Yaskawa INFORM job: A_NAIHAN_0617_1_PAINT_1.JBI

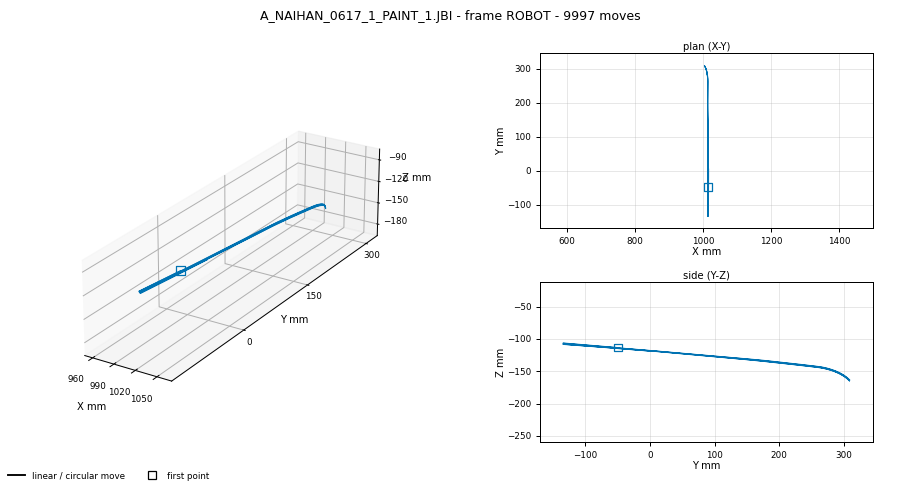
[picture p0: tool path of A_NAIHAN_0617_1_PAINT_1.JBI in frame ROBOT, 9997 of 9997 moves have a stored position in this frame; points joined in program order, loops and branches not executed]
/JOB
//NAME A_NAIHAN_0617_1_PAINT1
//POS
///NPOS 9997,0,0,0,0,0
///TOOL 1
///USER 0
///POSTYPE ROBOT
///RECTAN
///RCONF 0,0,0,0,1,0,0,0,0,0,0,0,0,0,0,0,0,0,0,0,0,0,0,0
C00000=1013.173,-49.105,-113.230,-28.110,44.378,-33.833
C00001=1013.171,-49.416,-113.204,-28.117,44.440,-33.820
C00002=1013.169,-49.806,-113.172,-28.126,44.517,-33.803
C00003=1013.167,-50.039,-113.152,-28.131,44.563,-33.794
C00004=1013.166,-50.273,-113.134,-28.136,44.610,-33.784
C00005=1013.165,-50.506,-113.114,-28.141,44.658,-33.775
C00006=1013.163,-50.741,-113.095,-28.147,44.706,-33.765
C00007=1013.162,-50.974,-113.075,-28.152,44.754,-33.754
C00008=1013.160,-51.207,-113.056,-28.157,44.802,-33.745
C00009=1013.160,-51.442,-113.037,-28.163,44.851,-33.735
C00010=1013.158,-51.675,-113.017,-28.168,44.899,-33.725
C00011=1013.156,-51.909,-112.998,-28.173,44.948,-33.715
C00012=1013.155,-52.143,-112.978,-28.179,44.998,-33.705
C00013=1013.154,-52.376,-112.959,-28.184,45.047,-33.695
C00014=1013.153,-52.610,-112.940,-28.189,45.097,-33.683
C00015=1013.151,-52.843,-112.921,-28.195,45.148,-33.674
C00016=1013.150,-53.077,-112.901,-28.200,45.199,-33.663
C00017=1013.148,-53.311,-112.882,-28.206,45.249,-33.653
C00018=1013.147,-53.544,-112.863,-28.212,45.300,-33.643
C00019=1013.146,-53.778,-112.844,-28.217,45.351,-33.632
C00020=1013.144,-54.011,-112.825,-28.223,45.403,-33.622
C00021=1013.143,-54.245,-112.804,-28.228,45.455,-33.612
C00022=1013.141,-54.479,-112.786,-28.234,45.507,-33.600
C00023=1013.140,-54.712,-112.766,-28.240,45.559,-33.590
C00024=1013.138,-54.946,-112.747,-28.245,45.612,-33.579
C00025=1013.137,-55.179,-112.728,-28.251,45.666,-33.568
C00026=1013.136,-55.414,-112.708,-28.257,45.718,-33.557
C00027=1013.134,-55.647,-112.689,-28.262,45.772,-33.547
C00028=1013.133,-55.881,-112.670,-28.268,45.825,-33.536
C00029=1013.131,-56.114,-112.651,-28.274,45.881,-33.525
C00030=1013.129,-56.348,-112.631,-28.280,45.934,-33.514
C00031=1013.129,-56.582,-112.612,-28.286,45.989,-33.503
C00032=1013.126,-56.816,-112.592,-28.292,46.045,-33.492
C00033=1013.125,-57.050,-112.573,-28.298,46.100,-33.480
C00034=1013.124,-57.284,-112.554,-28.304,46.156,-33.470
C00035=1013.122,-57.518,-112.534,-28.309,46.211,-33.459
C00036=1013.120,-57.753,-112.515,-28.315,46.268,-33.447
C00037=1013.119,-57.988,-112.495,-28.321,46.324,-33.437
C00038=1013.117,-58.222,-112.476,-28.328,46.382,-33.426
C00039=1013.116,-58.457,-112.457,-28.334,46.439,-33.414
C00040=1013.114,-58.693,-112.437,-28.340,46.496,-33.403
C00041=1013.113,-58.928,-112.418,-28.346,46.555,-33.390
C00042=1013.111,-59.163,-112.399,-28.352,46.614,-33.380
C00043=1013.110,-59.400,-112.379,-28.358,46.672,-33.368
C00044=1013.108,-59.635,-112.359,-28.364,46.732,-33.356
C00045=1013.107,-59.871,-112.340,-28.371,46.791,-33.345
C00046=1013.105,-60.108,-112.321,-28.377,46.850,-33.333
C00047=1013.103,-60.344,-112.301,-28.383,46.911,-33.322
C00048=1013.102,-60.581,-112.282,-28.390,46.972,-33.310
C00049=1013.101,-60.818,-112.262,-28.396,47.033,-33.298
C00050=1013.099,-61.055,-112.242,-28.402,47.093,-33.287
C00051=1013.097,-61.292,-112.222,-28.409,47.154,-33.275
C00052=1013.096,-61.529,-112.203,-28.415,47.217,-33.262
C00053=1013.094,-61.766,-112.183,-28.422,47.279,-33.251
C00054=1013.092,-62.005,-112.163,-28.428,47.341,-33.238
C00055=1013.090,-62.242,-112.144,-28.435,47.404,-33.227
C00056=1013.089,-62.480,-112.124,-28.441,47.467,-33.215
C00057=1013.087,-62.719,-112.104,-28.448,47.530,-33.203
C00058=1013.085,-62.957,-112.085,-28.455,47.595,-33.190
C00059=1013.083,-63.196,-112.065,-28.461,47.659,-33.178
C00060=1013.082,-63.434,-112.045,-28.468,47.723,-33.167
C00061=1013.080,-63.673,-112.025,-28.475,47.789,-33.155
C00062=1013.078,-63.913,-112.006,-28.481,47.854,-33.142
C00063=1013.077,-64.151,-111.986,-28.488,47.919,-33.130
C00064=1013.075,-64.391,-111.966,-28.495,47.985,-33.118
C00065=1013.073,-64.630,-111.946,-28.502,48.051,-33.105
C00066=1013.072,-64.870,-111.927,-28.508,48.117,-33.093
C00067=1013.070,-65.109,-111.907,-28.515,48.185,-33.081
C00068=1013.068,-65.349,-111.887,-28.522,48.252,-33.068
C00069=1013.067,-65.589,-111.867,-28.529,48.319,-33.056
C00070=1013.065,-65.829,-111.848,-28.536,48.387,-33.043
C00071=1013.062,-66.069,-111.827,-28.543,48.456,-33.030
C00072=1013.061,-66.309,-111.807,-28.550,48.524,-33.019
C00073=1013.059,-66.549,-111.787,-28.557,48.593,-33.005
C00074=1013.057,-66.790,-111.767,-28.564,48.662,-32.993
C00075=1013.056,-67.030,-111.747,-28.571,48.732,-32.980
C00076=1013.054,-67.270,-111.728,-28.578,48.802,-32.968
C00077=1013.052,-67.511,-111.707,-28.585,48.871,-32.956
C00078=1013.050,-67.752,-111.688,-28.593,48.941,-32.944
C00079=1013.049,-67.992,-111.668,-28.600,49.012,-32.931
C00080=1013.046,-68.233,-111.648,-28.607,49.083,-32.918
C00081=1013.044,-68.473,-111.628,-28.614,49.155,-32.905
C00082=1013.043,-68.713,-111.608,-28.621,49.227,-32.893
C00083=1013.040,-68.954,-111.588,-28.629,49.298,-32.880
C00084=1013.039,-69.195,-111.568,-28.636,49.371,-32.869
C00085=1013.037,-69.435,-111.549,-28.643,49.443,-32.855
C00086=1013.036,-69.676,-111.528,-28.650,49.516,-32.842
C00087=1013.033,-69.917,-111.509,-28.658,49.589,-32.830
C00088=1013.031,-70.158,-111.488,-28.665,49.662,-32.818
C00089=1013.030,-70.398,-111.469,-28.673,49.736,-32.805
C00090=1013.028,-70.639,-111.448,-28.680,49.811,-32.792
C00091=1013.026,-70.880,-111.429,-28.688,49.884,-32.779
C00092=1013.024,-71.110,-111.409,-28.695,49.956,-32.767
C00093=1013.022,-71.340,-111.390,-28.702,50.028,-32.756
C00094=1013.020,-71.601,-111.369,-28.710,50.110,-32.742
C00095=1013.019,-71.842,-111.349,-28.718,50.185,-32.729
C00096=1013.016,-72.082,-111.329,-28.725,50.261,-32.717
C00097=1013.014,-72.323,-111.309,-28.733,50.338,-32.703
C00098=1013.013,-72.563,-111.289,-28.741,50.414,-32.691
C00099=1013.010,-72.804,-111.269,-28.748,50.491,-32.678
C00100=1013.009,-73.044,-111.250,-28.756,50.567,-32.667
C00101=1013.007,-73.284,-111.229,-28.764,50.644,-32.653
C00102=1013.005,-73.524,-111.209,-28.771,50.722,-32.641
C00103=1013.003,-73.764,-111.189,-28.779,50.799,-32.628
C00104=1013.000,-74.004,-111.169,-28.787,50.879,-32.615
C00105=1012.999,-74.244,-111.149,-28.795,50.956,-32.603
C00106=1012.997,-74.484,-111.130,-28.803,51.036,-32.590
C00107=1012.995,-74.724,-111.109,-28.810,51.114,-32.578
C00108=1012.993,-74.964,-111.090,-28.818,51.193,-32.565
C00109=1012.991,-75.204,-111.070,-28.826,51.273,-32.553
C00110=1012.989,-75.443,-111.050,-28.834,51.353,-32.541
C00111=1012.987,-75.684,-111.030,-28.842,51.434,-32.527
C00112=1012.985,-75.924,-111.009,-28.850,51.514,-32.515
C00113=1012.983,-76.163,-110.990,-28.858,51.595,-32.502
C00114=1012.981,-76.403,-110.970,-28.866,51.675,-32.490
C00115=1012.979,-76.643,-110.950,-28.874,51.756,-32.478
C00116=1012.977,-76.882,-110.930,-28.882,51.838,-32.466
C00117=1012.975,-77.122,-110.910,-28.890,51.920,-32.454
C00118=1012.973,-77.360,-110.891,-28.899,52.002,-32.442
C00119=1012.971,-77.599,-110.871,-28.907,52.084,-32.428
C00120=1012.969,-77.839,-110.850,-28.915,52.167,-32.417
C00121=1012.967,-78.077,-110.831,-28.923,52.249,-32.403
C00122=1012.965,-78.316,-110.810,-28.931,52.333,-32.391
C00123=1012.963,-78.555,-110.791,-28.940,52.416,-32.381
C00124=1012.961,-78.794,-110.771,-28.948,52.499,-32.368
C00125=1012.959,-79.032,-110.751,-28.956,52.584,-32.355
C00126=1012.957,-79.271,-110.732,-28.965,52.668,-32.343
C00127=1012.955,-79.509,-110.711,-28.973,52.752,-32.332
C00128=1012.953,-79.747,-110.692,-28.981,52.837,-32.319
C00129=1012.951,-79.985,-110.672,-28.990,52.921,-32.308
C00130=1012.949,-80.222,-110.652,-28.998,53.006,-32.295
C00131=1012.947,-80.460,-110.632,-29.007,53.092,-32.283
C00132=1012.945,-80.697,-110.613,-29.015,53.177,-32.271
C00133=1012.943,-80.934,-110.593,-29.024,53.263,-32.259
C00134=1012.941,-81.169,-110.573,-29.032,53.348,-32.248
C00135=1012.939,-81.406,-110.554,-29.041,53.434,-32.236
C00136=1012.937,-81.643,-110.534,-29.049,53.520,-32.225
C00137=1012.935,-81.880,-110.514,-29.058,53.607,-32.213
C00138=1012.933,-82.117,-110.495,-29.067,53.695,-32.201
C00139=1012.930,-82.354,-110.475,-29.075,53.782,-32.190
C00140=1012.928,-82.591,-110.455,-29.084,53.870,-32.178
C00141=1012.927,-82.827,-110.435,-29.093,53.957,-32.166
C00142=1012.924,-83.062,-110.416,-29.102,54.045,-32.156
C00143=1012.922,-83.298,-110.395,-29.110,54.133,-32.144
C00144=1012.921,-83.535,-110.376,-29.119,54.222,-32.132
C00145=1012.918,-83.770,-110.357,-29.128,54.310,-32.122
C00146=1012.916,-84.002,-110.337,-29.137,54.397,-32.110
C00147=1012.914,-84.234,-110.318,-29.146,54.485,-32.100
C00148=1012.912,-84.468,-110.298,-29.155,54.574,-32.089
C00149=1012.910,-84.708,-110.278,-29.164,54.666,-32.077
C00150=1012.908,-84.964,-110.257,-29.174,54.764,-32.066
C00151=1012.905,-85.239,-110.234,-29.184,54.869,-32.052
C00152=1012.903,-85.524,-110.210,-29.195,54.978,-32.039
C00153=1012.900,-85.807,-110.187,-29.206,55.087,-32.027
C00154=1012.898,-86.076,-110.164,-29.217,55.192,-32.014
C00155=1012.895,-86.327,-110.142,-29.227,55.290,-32.003
C00156=1012.894,-86.561,-110.123,-29.236,55.382,-31.992
C00157=1012.892,-86.793,-110.104,-29.245,55.471,-31.982
C00158=1012.889,-87.101,-110.078,-29.258,55.593,-31.968
C00159=1012.886,-87.464,-110.048,-29.272,55.737,-31.952
C00160=1012.884,-87.683,-110.030,-29.281,55.823,-31.942
C00161=1012.882,-87.899,-110.012,-29.290,55.908,-31.933
C00162=1012.880,-88.115,-109.993,-29.299,55.995,-31.924
C00163=1012.878,-88.341,-109.975,-29.308,56.085,-31.914
C00164=1012.875,-88.568,-109.956,-29.317,56.176,-31.905
C00165=1012.874,-88.801,-109.936,-29.327,56.270,-31.895
C00166=1012.871,-89.068,-109.913,-29.338,56.377,-31.883
C00167=1012.869,-89.365,-109.889,-29.351,56.498,-31.872
C00168=1012.866,-89.673,-109.863,-29.364,56.623,-31.858
C00169=1012.863,-89.974,-109.838,-29.376,56.745,-31.846
C00170=1012.861,-90.252,-109.814,-29.388,56.859,-31.835
C00171=1012.857,-90.648,-109.782,-29.406,57.022,-31.820
C00172=1012.855,-90.945,-109.757,-29.418,57.144,-31.807
C00173=1012.853,-91.195,-109.736,-29.429,57.248,-31.797
C00174=1012.851,-91.427,-109.716,-29.439,57.344,-31.789
C00175=1012.849,-91.658,-109.697,-29.449,57.441,-31.780
C00176=1012.847,-91.889,-109.677,-29.460,57.536,-31.771
C00177=1012.844,-92.120,-109.658,-29.470,57.633,-31.762
C00178=1012.842,-92.352,-109.639,-29.480,57.730,-31.753
C00179=1012.840,-92.582,-109.620,-29.491,57.828,-31.745
C00180=1012.838,-92.812,-109.600,-29.501,57.925,-31.737
C00181=1012.837,-93.042,-109.581,-29.511,58.022,-31.728
C00182=1012.834,-93.271,-109.561,-29.522,58.119,-31.721
C00183=1012.831,-93.501,-109.542,-29.533,58.217,-31.713
C00184=1012.830,-93.730,-109.523,-29.543,58.315,-31.703
C00185=1012.828,-93.959,-109.504,-29.554,58.412,-31.696
C00186=1012.826,-94.188,-109.485,-29.565,58.510,-31.689
C00187=1012.824,-94.416,-109.465,-29.575,58.608,-31.681
C00188=1012.821,-94.643,-109.447,-29.586,58.706,-31.674
C00189=1012.819,-94.871,-109.427,-29.597,58.805,-31.666
C00190=1012.817,-95.097,-109.408,-29.608,58.902,-31.659
C00191=1012.816,-95.323,-109.389,-29.619,59.001,-31.652
C00192=1012.814,-95.549,-109.370,-29.630,59.100,-31.645
C00193=1012.812,-95.774,-109.351,-29.641,59.197,-31.638
C00194=1012.810,-95.999,-109.332,-29.652,59.297,-31.632
C00195=1012.807,-96.224,-109.313,-29.663,59.395,-31.625
C00196=1012.806,-96.448,-109.294,-29.674,59.494,-31.618
C00197=1012.804,-96.673,-109.275,-29.685,59.592,-31.611
C00198=1012.802,-96.896,-109.257,-29.697,59.692,-31.605
C00199=1012.799,-97.121,-109.238,-29.708,59.791,-31.599
C00200=1012.798,-97.345,-109.219,-29.720,59.890,-31.594
C00201=1012.796,-97.568,-109.200,-29.732,59.990,-31.589
C00202=1012.794,-97.791,-109.182,-29.743,60.090,-31.582
C00203=1012.792,-98.015,-109.162,-29.755,60.189,-31.577
C00204=1012.790,-98.239,-109.144,-29.766,60.289,-31.571
C00205=1012.788,-98.462,-109.125,-29.778,60.390,-31.566
C00206=1012.786,-98.686,-109.106,-29.790,60.491,-31.560
C00207=1012.784,-98.910,-109.088,-29.802,60.591,-31.555
C00208=1012.782,-99.134,-109.068,-29.814,60.693,-31.551
C00209=1012.780,-99.358,-109.050,-29.827,60.795,-31.545
C00210=1012.778,-99.582,-109.030,-29.839,60.896,-31.542
C00211=1012.776,-99.807,-109.011,-29.851,60.999,-31.537
C00212=1012.774,-100.080,-108.988,-29.866,61.123,-31.531
C00213=1012.770,-100.484,-108.955,-29.889,61.308,-31.523
C00214=1012.768,-100.710,-108.936,-29.902,61.411,-31.520
C00215=1012.766,-100.937,-108.916,-29.915,61.515,-31.515
C00216=1012.764,-101.163,-108.898,-29.928,61.620,-31.512
C00217=1012.762,-101.391,-108.878,-29.942,61.725,-31.509
C00218=1012.760,-101.619,-108.859,-29.955,61.831,-31.505
C00219=1012.758,-101.846,-108.839,-29.968,61.937,-31.501
C00220=1012.756,-102.075,-108.820,-29.982,62.042,-31.499
C00221=1012.754,-102.303,-108.801,-29.995,62.148,-31.496
C00222=1012.752,-102.533,-108.782,-30.009,62.256,-31.492
C00223=1012.750,-102.762,-108.762,-30.023,62.363,-31.491
C00224=1012.748,-102.992,-108.743,-30.037,62.471,-31.488
C00225=1012.746,-103.221,-108.724,-30.052,62.577,-31.486
C00226=1012.745,-103.451,-108.704,-30.066,62.686,-31.484
C00227=1012.742,-103.681,-108.685,-30.080,62.794,-31.482
C00228=1012.740,-103.912,-108.666,-30.095,62.903,-31.479
C00229=1012.738,-104.142,-108.646,-30.110,63.012,-31.479
C00230=1012.737,-104.372,-108.627,-30.125,63.121,-31.477
C00231=1012.734,-104.603,-108.607,-30.140,63.231,-31.476
C00232=1012.732,-104.835,-108.588,-30.155,63.341,-31.475
C00233=1012.730,-105.066,-108.568,-30.170,63.451,-31.474
C00234=1012.729,-105.296,-108.549,-30.186,63.561,-31.474
C00235=1012.727,-105.528,-108.529,-30.201,63.671,-31.474
C00236=1012.724,-105.760,-108.509,-30.217,63.783,-31.473
C00237=1012.722,-105.991,-108.489,-30.233,63.893,-31.475
C00238=1012.721,-106.223,-108.470,-30.249,64.005,-31.475
C00239=1012.718,-106.458,-108.450,-30.266,64.119,-31.476
C00240=1012.716,-106.700,-108.430,-30.283,64.236,-31.476
C00241=1012.714,-106.952,-108.408,-30.301,64.358,-31.478
C00242=1012.712,-107.215,-108.386,-30.320,64.486,-31.480
C00243=1012.710,-107.485,-108.363,-30.340,64.617,-31.481
C00244=1012.708,-107.760,-108.340,-30.360,64.750,-31.484
C00245=1012.705,-108.036,-108.317,-30.381,64.885,-31.486
C00246=1012.703,-108.311,-108.294,-30.402,65.020,-31.489
C00247=1012.701,-108.579,-108.270,-30.422,65.151,-31.492
C00248=1012.698,-108.839,-108.249,-30.442,65.279,-31.494
C00249=1012.697,-109.090,-108.227,-30.462,65.403,-31.498
C00250=1012.694,-109.330,-108.207,-30.482,65.521,-31.504
C00251=1012.693,-109.564,-108.188,-30.501,65.636,-31.508
C00252=1012.692,-109.795,-108.168,-30.519,65.751,-31.512
C00253=1012.689,-110.026,-108.148,-30.538,65.866,-31.517
C00254=1012.687,-110.258,-108.129,-30.558,65.981,-31.522
C00255=1012.686,-110.489,-108.109,-30.577,66.096,-31.527
C00256=1012.684,-110.721,-108.089,-30.597,66.212,-31.532
C00257=1012.682,-110.952,-108.069,-30.617,66.327,-31.538
C00258=1012.680,-111.183,-108.050,-30.637,66.444,-31.544
C00259=1012.678,-111.483,-108.024,-30.664,66.593,-31.553
C00260=1012.675,-111.878,-107.991,-30.699,66.792,-31.564
C00261=1012.672,-112.109,-107.971,-30.720,66.908,-31.572
C00262=1012.671,-112.340,-107.952,-30.741,67.024,-31.579
C00263=1012.669,-112.571,-107.932,-30.763,67.142,-31.587
C00264=1012.667,-112.803,-107.913,-30.784,67.259,-31.596
C00265=1012.666,-113.035,-107.893,-30.807,67.377,-31.604
C00266=1012.663,-113.266,-107.873,-30.829,67.494,-31.615
C00267=1012.662,-113.497,-107.854,-30.852,67.612,-31.624
C00268=1012.660,-113.728,-107.834,-30.875,67.730,-31.634
C00269=1012.658,-113.959,-107.815,-30.898,67.848,-31.644
C00270=1012.657,-114.190,-107.795,-30.922,67.965,-31.654
C00271=1012.655,-114.422,-107.775,-30.945,68.085,-31.665
C00272=1012.653,-114.653,-107.756,-30.970,68.203,-31.677
C00273=1012.651,-114.885,-107.736,-30.994,68.322,-31.687
C00274=1012.650,-115.115,-107.716,-31.018,68.441,-31.699
C00275=1012.648,-115.347,-107.697,-31.044,68.561,-31.713
C00276=1012.646,-115.578,-107.677,-31.070,68.680,-31.727
C00277=1012.644,-115.809,-107.658,-31.095,68.800,-31.738
C00278=1012.642,-116.040,-107.637,-31.121,68.919,-31.753
C00279=1012.641,-116.271,-107.619,-31.148,69.039,-31.769
C00280=1012.639,-116.503,-107.598,-31.175,69.160,-31.783
C00281=1012.637,-116.734,-107.579,-31.202,69.281,-31.798
C00282=1012.636,-116.965,-107.559,-31.230,69.400,-31.814
C00283=1012.635,-117.196,-107.540,-31.258,69.521,-31.830
C00284=1012.632,-117.427,-107.520,-31.286,69.642,-31.848
C00285=1012.631,-117.659,-107.500,-31.314,69.764,-31.863
C00286=1012.629,-117.890,-107.481,-31.344,69.885,-31.881
C00287=1012.628,-118.121,-107.461,-31.374,70.006,-31.900
C00288=1012.626,-118.352,-107.441,-31.404,70.128,-31.918
C00289=1012.624,-118.584,-107.422,-31.434,70.250,-31.937
C00290=1012.623,-118.814,-107.402,-31.465,70.373,-31.958
C00291=1012.621,-119.046,-107.383,-31.496,70.495,-31.977
C00292=1012.619,-119.277,-107.363,-31.529,70.617,-31.999
C00293=1012.618,-119.507,-107.343,-31.562,70.740,-32.021
C00294=1012.616,-119.739,-107.324,-31.593,70.862,-32.041
C00295=1012.615,-119.970,-107.303,-31.628,70.985,-32.066
C00296=1012.613,-120.201,-107.284,-31.662,71.109,-32.089
C00297=1012.611,-120.432,-107.265,-31.696,71.232,-32.112
C00298=1012.610,-120.663,-107.245,-31.731,71.356,-32.138
C00299=1012.608,-120.894,-107.225,-31.766,71.479,-32.162
C00300=1012.607,-121.126,-107.206,-31.803,71.603,-32.189
C00301=1012.605,-121.356,-107.186,-31.839,71.728,-32.215
C00302=1012.604,-121.588,-107.167,-31.877,71.851,-32.243
C00303=1012.602,-121.885,-107.141,-31.925,72.012,-32.278
C00304=1012.600,-122.280,-107.107,-31.992,72.225,-32.329
C00305=1012.598,-122.511,-107.087,-32.033,72.351,-32.360
///RCONF 0,0,0,0,0,0,0,0,0,0,0,0,0,0,0,0,0,0,0,0,0,0,0,0
C00306=1012.597,-122.742,-107.068,-32.073,72.475,-32.390
C00307=1012.595,-122.973,-107.048,-32.114,72.600,-32.423
C00308=1012.594,-123.204,-107.029,-32.156,72.726,-32.454
C00309=1012.592,-123.435,-107.009,-32.199,72.851,-32.489
C00310=1012.591,-123.666,-106.990,-32.242,72.976,-32.522
C00311=1012.589,-123.897,-106.970,-32.286,73.102,-32.557
C00312=1012.588,-124.128,-106.951,-32.331,73.229,-32.594
C00313=1012.586,-124.360,-106.930,-32.377,73.354,-32.630
C00314=1012.585,-124.590,-106.911,-32.424,73.480,-32.669
C00315=1012.584,-124.822,-106.891,-32.471,73.606,-32.707
C00316=1012.582,-125.052,-106.872,-32.519,73.733,-32.746
C00317=1012.581,-125.284,-106.852,-32.568,73.859,-32.788
C00318=1012.580,-125.514,-106.832,-32.618,73.986,-32.830
C00319=1012.578,-125.745,-106.813,-32.669,74.113,-32.872
C00320=1012.577,-125.976,-106.793,-32.720,74.239,-32.915
C00321=1012.575,-126.207,-106.774,-32.773,74.366,-32.960
C00322=1012.574,-126.438,-106.754,-32.827,74.493,-33.007
C00323=1012.573,-126.669,-106.734,-32.882,74.620,-33.054
C00324=1012.571,-126.900,-106.715,-32.939,74.747,-33.103
C00325=1012.570,-127.132,-106.695,-32.995,74.874,-33.151
C00326=1012.569,-127.362,-106.675,-33.053,75.002,-33.201
C00327=1012.567,-127.592,-106.655,-33.113,75.129,-33.255
C00328=1012.566,-127.824,-106.636,-33.173,75.257,-33.308
C00329=1012.565,-128.055,-106.616,-33.235,75.385,-33.363
C00330=1012.564,-128.285,-106.597,-33.297,75.514,-33.417
C00331=1012.562,-128.517,-106.577,-33.361,75.641,-33.474
C00332=1012.562,-128.748,-106.557,-33.427,75.770,-33.535
C00333=1012.560,-128.978,-106.538,-33.493,75.898,-33.593
C00334=1012.559,-129.210,-106.518,-33.562,76.027,-33.655
C00335=1012.558,-129.440,-106.498,-33.633,76.155,-33.721
C00336=1012.556,-129.671,-106.479,-33.704,76.284,-33.786
C00337=1012.555,-129.902,-106.459,-33.775,76.413,-33.849
C00338=1012.554,-130.134,-106.439,-33.850,76.541,-33.918
C00339=1012.553,-130.364,-106.419,-33.926,76.670,-33.988
C00340=1012.552,-130.595,-106.401,-34.004,76.800,-34.061
C00341=1012.551,-130.825,-106.381,-34.084,76.929,-34.135
C00342=1012.550,-131.057,-106.361,-34.164,77.058,-34.209
C00343=1012.549,-131.288,-106.341,-34.248,77.188,-34.288
C00344=1012.547,-131.603,-106.314,-34.364,77.365,-34.396
C00345=1012.545,-131.980,-106.283,-34.508,77.577,-34.531
C00346=1012.545,-132.211,-106.263,-34.600,77.706,-34.619
C00347=1012.543,-132.443,-106.243,-34.693,77.837,-34.706
C00348=1012.542,-132.673,-106.224,-34.789,77.966,-34.798
C00349=1012.541,-132.904,-106.204,-34.887,78.096,-34.891
C00350=1012.540,-133.135,-106.184,-34.989,78.227,-34.988
C00351=1012.539,-133.366,-106.165,-35.090,78.357,-35.084
C00352=1012.538,-133.596,-106.145,-35.195,78.487,-35.184
C00353=1012.537,-133.827,-106.126,-35.304,78.618,-35.290
C00354=1012.536,-134.058,-106.106,-35.416,78.749,-35.397
///RCONF 0,0,0,0,1,0,0,0,0,0,0,0,0,0,0,0,0,0,0,0,0,0,0,0
C00355=1012.642,-134.083,-106.545,-31.212,69.079,-31.891
C00356=1012.643,-133.853,-106.565,-31.181,68.940,-31.876
C00357=1012.645,-133.622,-106.584,-31.151,68.800,-31.861
C00358=1012.648,-133.391,-106.604,-31.121,68.662,-31.846
C00359=1012.649,-133.161,-106.623,-31.091,68.523,-31.831
C00360=1012.652,-132.930,-106.643,-31.063,68.383,-31.818
C00361=1012.654,-132.698,-106.662,-31.034,68.245,-31.804
C00362=1012.655,-132.468,-106.681,-31.006,68.107,-31.792
C00363=1012.658,-132.237,-106.701,-30.978,67.968,-31.779
C00364=1012.659,-132.006,-106.722,-30.950,67.831,-31.767
C00365=1012.662,-131.775,-106.742,-30.923,67.692,-31.756
C00366=1012.663,-131.544,-106.760,-30.896,67.555,-31.745
C00367=1012.665,-131.313,-106.780,-30.870,67.417,-31.736
C00368=1012.668,-131.082,-106.800,-30.844,67.280,-31.727
C00369=1012.670,-130.851,-106.820,-30.818,67.142,-31.717
C00370=1012.672,-130.621,-106.839,-30.793,67.005,-31.707
C00371=1012.674,-130.390,-106.858,-30.768,66.868,-31.700
C00372=1012.676,-130.167,-106.878,-30.744,66.735,-31.693
C00373=1012.678,-129.928,-106.898,-30.719,66.594,-31.686
C00374=1012.680,-129.698,-106.917,-30.695,66.458,-31.678
C00375=1012.682,-129.467,-106.937,-30.671,66.321,-31.672
C00376=1012.685,-129.235,-106.956,-30.648,66.185,-31.666
C00377=1012.687,-129.005,-106.976,-30.624,66.049,-31.659
C00378=1012.690,-128.774,-106.995,-30.602,65.913,-31.654
C00379=1012.692,-128.543,-107.015,-30.579,65.778,-31.650
C00380=1012.694,-128.312,-107.035,-30.556,65.641,-31.645
C00381=1012.696,-128.081,-107.054,-30.534,65.506,-31.641
C00382=1012.698,-127.850,-107.074,-30.513,65.370,-31.638
C00383=1012.700,-127.619,-107.094,-30.491,65.236,-31.635
C00384=1012.702,-127.388,-107.113,-30.470,65.100,-31.633
C00385=1012.704,-127.157,-107.132,-30.449,64.965,-31.629
C00386=1012.707,-126.926,-107.152,-30.428,64.831,-31.627
C00387=1012.709,-126.695,-107.172,-30.407,64.697,-31.626
C00388=1012.711,-126.465,-107.191,-30.387,64.562,-31.624
C00389=1012.714,-126.234,-107.211,-30.366,64.428,-31.623
C00390=1012.716,-126.003,-107.230,-30.347,64.293,-31.622
C00391=1012.718,-125.772,-107.250,-30.327,64.160,-31.623
C00392=1012.720,-125.541,-107.270,-30.307,64.026,-31.622
C00393=1012.723,-125.310,-107.289,-30.288,63.892,-31.623
C00394=1012.725,-125.078,-107.308,-30.269,63.759,-31.623
C00395=1012.728,-124.848,-107.328,-30.250,63.626,-31.624
C00396=1012.730,-124.617,-107.348,-30.231,63.493,-31.625
C00397=1012.732,-124.386,-107.367,-30.213,63.360,-31.627
C00398=1012.735,-124.155,-107.387,-30.194,63.227,-31.629
C00399=1012.737,-123.923,-107.406,-30.176,63.094,-31.631
C00400=1012.739,-123.692,-107.426,-30.158,62.961,-31.633
C00401=1012.742,-123.462,-107.445,-30.140,62.830,-31.636
C00402=1012.744,-123.231,-107.465,-30.122,62.697,-31.640
C00403=1012.746,-122.999,-107.484,-30.104,62.565,-31.642
C00404=1012.749,-122.769,-107.504,-30.087,62.434,-31.645
C00405=1012.752,-122.538,-107.523,-30.070,62.303,-31.650
C00406=1012.754,-122.307,-107.543,-30.053,62.170,-31.655
C00407=1012.756,-122.075,-107.562,-30.035,62.040,-31.658
C00408=1012.758,-121.845,-107.582,-30.019,61.909,-31.663
C00409=1012.760,-121.614,-107.602,-30.002,61.777,-31.668
C00410=1012.764,-121.383,-107.621,-29.986,61.646,-31.674
C00411=1012.766,-121.152,-107.640,-29.969,61.516,-31.679
C00412=1012.768,-120.921,-107.660,-29.953,61.385,-31.685
C00413=1012.772,-120.573,-107.689,-29.929,61.189,-31.694
C00414=1012.776,-120.227,-107.719,-29.905,60.995,-31.703
C00415=1012.778,-119.996,-107.738,-29.889,60.866,-31.710
C00416=1012.781,-119.765,-107.758,-29.873,60.736,-31.717
C00417=1012.783,-119.534,-107.777,-29.858,60.606,-31.724
C00418=1012.785,-119.303,-107.797,-29.842,60.477,-31.732
C00419=1012.788,-119.072,-107.816,-29.827,60.348,-31.739
C00420=1012.790,-118.841,-107.835,-29.812,60.219,-31.748
C00421=1012.793,-118.610,-107.855,-29.797,60.091,-31.756
C00422=1012.796,-118.378,-107.875,-29.782,59.962,-31.765
C00423=1012.799,-118.148,-107.894,-29.767,59.834,-31.774
C00424=1012.801,-117.916,-107.913,-29.752,59.705,-31.782
C00425=1012.803,-117.685,-107.933,-29.737,59.577,-31.791
C00426=1012.806,-117.455,-107.952,-29.723,59.450,-31.801
C00427=1012.808,-117.223,-107.972,-29.708,59.323,-31.809
C00428=1012.811,-116.991,-107.992,-29.694,59.195,-31.820
C00429=1012.814,-116.761,-108.011,-29.679,59.068,-31.828
C00430=1012.816,-116.529,-108.030,-29.665,58.941,-31.839
C00431=1012.818,-116.298,-108.050,-29.651,58.814,-31.849
C00432=1012.821,-116.068,-108.069,-29.637,58.688,-31.860
C00433=1012.824,-115.836,-108.089,-29.623,58.562,-31.870
C00434=1012.826,-115.605,-108.108,-29.609,58.436,-31.882
C00435=1012.829,-115.373,-108.127,-29.596,58.310,-31.893
C00436=1012.831,-115.143,-108.147,-29.582,58.185,-31.904
C00437=1012.834,-114.911,-108.167,-29.568,58.059,-31.916
C00438=1012.837,-114.680,-108.185,-29.555,57.934,-31.927
C00439=1012.839,-114.449,-108.205,-29.541,57.810,-31.938
C00440=1012.842,-114.217,-108.226,-29.528,57.685,-31.950
C00441=1012.845,-113.986,-108.244,-29.514,57.561,-31.962
C00442=1012.847,-113.755,-108.264,-29.501,57.437,-31.974
C00443=1012.850,-113.524,-108.282,-29.488,57.313,-31.988
C00444=1012.853,-113.292,-108.303,-29.475,57.189,-32.000
C00445=1012.855,-113.061,-108.322,-29.462,57.066,-32.013
C00446=1012.858,-112.830,-108.341,-29.449,56.943,-32.026
C00447=1012.861,-112.598,-108.361,-29.436,56.820,-32.040
C00448=1012.863,-112.367,-108.380,-29.423,56.697,-32.053
C00449=1012.866,-112.136,-108.399,-29.410,56.574,-32.066
C00450=1012.868,-111.904,-108.419,-29.398,56.452,-32.080
C00451=1012.871,-111.673,-108.438,-29.384,56.330,-32.092
C00452=1012.873,-111.442,-108.457,-29.372,56.208,-32.107
C00453=1012.876,-111.210,-108.477,-29.359,56.086,-32.121
C00454=1012.879,-110.979,-108.496,-29.347,55.966,-32.136
C00455=1012.882,-110.747,-108.516,-29.334,55.845,-32.149
C00456=1012.886,-110.380,-108.547,-29.315,55.653,-32.173
C00457=1012.890,-110.053,-108.573,-29.297,55.483,-32.193
C00458=1012.893,-109.822,-108.593,-29.285,55.363,-32.208
C00459=1012.895,-109.590,-108.613,-29.273,55.243,-32.224
C00460=1012.898,-109.357,-108.633,-29.260,55.121,-32.238
C00461=1012.901,-109.117,-108.652,-29.247,54.998,-32.254
C00462=1012.904,-108.866,-108.673,-29.234,54.870,-32.270
C00463=1012.907,-108.606,-108.695,-29.221,54.736,-32.289
C00464=1012.910,-108.337,-108.717,-29.207,54.599,-32.306
C00465=1012.913,-108.064,-108.741,-29.193,54.458,-32.325
C00466=1012.917,-107.787,-108.764,-29.179,54.317,-32.346
C00467=1012.920,-107.512,-108.787,-29.164,54.177,-32.364
C00468=1012.923,-107.242,-108.809,-29.151,54.040,-32.385
C00469=1012.926,-106.979,-108.831,-29.137,53.907,-32.403
C00470=1012.929,-106.727,-108.852,-29.125,53.780,-32.421
C00471=1012.932,-106.484,-108.872,-29.112,53.657,-32.438
C00472=1012.935,-106.249,-108.892,-29.100,53.539,-32.456
C00473=1012.937,-106.018,-108.911,-29.089,53.423,-32.472
C00474=1012.940,-105.786,-108.930,-29.077,53.307,-32.490
C00475=1012.943,-105.555,-108.950,-29.065,53.191,-32.507
C00476=1012.945,-105.324,-108.969,-29.054,53.076,-32.524
C00477=1012.949,-105.093,-108.988,-29.042,52.961,-32.541
C00478=1012.951,-104.861,-109.007,-29.031,52.847,-32.559
C00479=1012.954,-104.630,-109.027,-29.019,52.732,-32.576
C00480=1012.957,-104.400,-109.046,-29.008,52.618,-32.595
C00481=1012.959,-104.169,-109.066,-28.997,52.504,-32.613
C00482=1012.961,-103.939,-109.085,-28.985,52.391,-32.630
C00483=1012.964,-103.708,-109.104,-28.974,52.278,-32.648
C00484=1012.967,-103.479,-109.123,-28.963,52.166,-32.666
C00485=1012.970,-103.248,-109.142,-28.951,52.053,-32.684
C00486=1012.973,-103.019,-109.162,-28.940,51.941,-32.702
C00487=1012.975,-102.789,-109.180,-28.929,51.829,-32.721
C00488=1012.979,-102.560,-109.199,-28.918,51.718,-32.739
C00489=1012.981,-102.331,-109.219,-28.907,51.607,-32.757
C00490=1012.984,-102.102,-109.238,-28.896,51.497,-32.776
C00491=1012.986,-101.874,-109.257,-28.884,51.386,-32.795
C00492=1012.989,-101.646,-109.275,-28.873,51.276,-32.814
C00493=1012.992,-101.418,-109.294,-28.863,51.168,-32.832
C00494=1012.995,-101.191,-109.313,-28.851,51.059,-32.850
C00495=1012.997,-100.964,-109.332,-28.841,50.949,-32.870
C00496=1013.000,-100.737,-109.351,-28.830,50.843,-32.889
C00497=1013.002,-100.511,-109.370,-28.819,50.734,-32.908
C00498=1013.005,-100.285,-109.388,-28.808,50.627,-32.926
C00499=1013.008,-100.060,-109.407,-28.797,50.520,-32.946
C00500=1013.010,-99.834,-109.426,-28.787,50.414,-32.965
C00501=1013.013,-99.610,-109.445,-28.776,50.309,-32.983
C00502=1013.016,-99.385,-109.463,-28.765,50.203,-33.003
C00503=1013.020,-99.061,-109.490,-28.750,50.051,-33.031
C00504=1013.024,-98.713,-109.518,-28.733,49.888,-33.061
C00505=1013.026,-98.489,-109.537,-28.723,49.784,-33.080
C00506=1013.029,-98.266,-109.556,-28.712,49.680,-33.100
C00507=1013.032,-98.042,-109.574,-28.702,49.577,-33.119
C00508=1013.034,-97.819,-109.593,-28.691,49.473,-33.138
C00509=1013.037,-97.595,-109.611,-28.680,49.370,-33.157
C00510=1013.040,-97.372,-109.630,-28.670,49.266,-33.178
C00511=1013.042,-97.148,-109.649,-28.660,49.165,-33.198
C00512=1013.045,-96.923,-109.667,-28.649,49.062,-33.217
C00513=1013.048,-96.700,-109.685,-28.638,48.959,-33.237
C00514=1013.050,-96.476,-109.703,-28.628,48.857,-33.257
C00515=1013.053,-96.251,-109.723,-28.618,48.756,-33.277
C00516=1013.056,-96.027,-109.741,-28.607,48.654,-33.297
C00517=1013.059,-95.801,-109.759,-28.597,48.552,-33.318
C00518=1013.060,-95.576,-109.778,-28.586,48.451,-33.337
C00519=1013.064,-95.350,-109.797,-28.575,48.349,-33.358
C00520=1013.066,-95.124,-109.816,-28.565,48.247,-33.378
C00521=1013.069,-94.897,-109.835,-28.554,48.145,-33.399
C00522=1013.072,-94.670,-109.853,-28.544,48.044,-33.419
C00523=1013.074,-94.443,-109.871,-28.533,47.943,-33.441
C00524=1013.076,-94.214,-109.891,-28.523,47.841,-33.462
C00525=1013.079,-93.986,-109.909,-28.512,47.741,-33.482
C00526=1013.082,-93.757,-109.929,-28.501,47.639,-33.503
C00527=1013.085,-93.529,-109.948,-28.491,47.538,-33.525
C00528=1013.087,-93.299,-109.966,-28.480,47.437,-33.545
C00529=1013.090,-93.069,-109.985,-28.470,47.336,-33.568
C00530=1013.092,-92.839,-110.004,-28.459,47.236,-33.589
C00531=1013.095,-92.608,-110.023,-28.448,47.135,-33.610
C00532=1013.098,-92.378,-110.043,-28.438,47.034,-33.632
C00533=1013.101,-92.148,-110.061,-28.427,46.935,-33.654
C00534=1013.104,-91.917,-110.080,-28.416,46.835,-33.675
C00535=1013.106,-91.685,-110.100,-28.406,46.735,-33.697
C00536=1013.109,-91.454,-110.119,-28.395,46.637,-33.718
C00537=1013.112,-91.223,-110.137,-28.384,46.536,-33.739
C00538=1013.114,-90.973,-110.158,-28.373,46.430,-33.762
C00539=1013.118,-90.675,-110.183,-28.360,46.303,-33.793
C00540=1013.123,-90.280,-110.215,-28.341,46.136,-33.829
C00541=1013.126,-90.001,-110.239,-28.329,46.019,-33.855
C00542=1013.129,-89.700,-110.263,-28.315,45.892,-33.884
C00543=1013.132,-89.392,-110.289,-28.301,45.763,-33.912
C00544=1013.136,-89.095,-110.312,-28.287,45.640,-33.941
C00545=1013.139,-88.828,-110.334,-28.275,45.529,-33.967
C00546=1013.142,-88.595,-110.353,-28.265,45.432,-33.990
C00547=1013.144,-88.368,-110.372,-28.254,45.338,-34.011
C00548=1013.147,-88.142,-110.392,-28.244,45.246,-34.032
C00549=1013.149,-87.925,-110.409,-28.234,45.157,-34.053
C00550=1013.152,-87.710,-110.426,-28.224,45.069,-34.073
C00551=1013.155,-87.492,-110.445,-28.215,44.980,-34.095
C00552=1013.157,-87.271,-110.463,-28.205,44.891,-34.116
C00553=1013.160,-87.048,-110.481,-28.195,44.800,-34.137
C00554=1013.162,-86.819,-110.500,-28.184,44.708,-34.159
C00555=1013.165,-86.588,-110.518,-28.174,44.614,-34.182
C00556=1013.169,-86.169,-110.553,-28.155,44.447,-34.222
C00557=1013.173,-85.834,-110.581,-28.140,44.313,-34.255
C00558=1013.176,-85.551,-110.604,-28.127,44.201,-34.281
C00559=1013.180,-85.266,-110.627,-28.114,44.088,-34.309
C00560=1013.183,-84.991,-110.650,-28.102,43.980,-34.335
C00561=1013.186,-84.736,-110.671,-28.091,43.880,-34.360
C00562=1013.188,-84.495,-110.691,-28.080,43.786,-34.383
C00563=1013.191,-84.262,-110.710,-28.069,43.695,-34.406
C00564=1013.193,-84.030,-110.729,-28.059,43.605,-34.429
C00565=1013.196,-83.796,-110.748,-28.049,43.515,-34.451
C00566=1013.198,-83.561,-110.767,-28.038,43.425,-34.474
C00567=1013.200,-83.325,-110.786,-28.028,43.333,-34.497
C00568=1013.204,-83.089,-110.806,-28.017,43.243,-34.519
C00569=1013.207,-82.853,-110.826,-28.007,43.153,-34.543
C00570=1013.209,-82.617,-110.844,-27.996,43.064,-34.565
C00571=1013.212,-82.382,-110.864,-27.986,42.974,-34.588
C00572=1013.214,-82.143,-110.883,-27.975,42.885,-34.610
C00573=1013.217,-81.907,-110.902,-27.965,42.796,-34.635
C00574=1013.219,-81.669,-110.922,-27.954,42.707,-34.656
C00575=1013.222,-81.433,-110.941,-27.944,42.619,-34.680
C00576=1013.224,-81.197,-110.961,-27.933,42.531,-34.702
C00577=1013.226,-80.960,-110.980,-27.923,42.443,-34.726
C00578=1013.229,-80.724,-110.999,-27.912,42.356,-34.748
C00579=1013.232,-80.487,-111.018,-27.902,42.269,-34.771
C00580=1013.235,-80.250,-111.038,-27.892,42.182,-34.794
C00581=1013.237,-80.011,-111.058,-27.881,42.095,-34.817
C00582=1013.239,-79.774,-111.078,-27.871,42.008,-34.840
C00583=1013.242,-79.536,-111.097,-27.860,41.922,-34.864
C00584=1013.245,-79.298,-111.116,-27.850,41.836,-34.886
C00585=1013.248,-79.059,-111.135,-27.839,41.750,-34.909
C00586=1013.249,-78.820,-111.155,-27.829,41.665,-34.932
C00587=1013.251,-78.582,-111.174,-27.818,41.579,-34.956
C00588=1013.254,-78.343,-111.194,-27.808,41.494,-34.978
C00589=1013.257,-78.104,-111.214,-27.798,41.410,-35.002
C00590=1013.259,-77.866,-111.233,-27.787,41.326,-35.024
C00591=1013.262,-77.627,-111.252,-27.777,41.242,-35.047
C00592=1013.264,-77.387,-111.272,-27.766,41.158,-35.071
C00593=1013.267,-77.148,-111.292,-27.756,41.074,-35.093
C00594=1013.270,-76.909,-111.311,-27.746,40.992,-35.116
C00595=1013.272,-76.669,-111.331,-27.735,40.907,-35.139
C00596=1013.274,-76.429,-111.350,-27.725,40.825,-35.162
C00597=1013.276,-76.190,-111.370,-27.715,40.744,-35.184
C00598=1013.280,-75.950,-111.389,-27.704,40.661,-35.207
C00599=1013.282,-75.711,-111.410,-27.694,40.579,-35.231
C00600=1013.284,-75.471,-111.428,-27.684,40.498,-35.253
C00601=1013.287,-75.230,-111.448,-27.673,40.417,-35.277
C00602=1013.289,-74.991,-111.467,-27.663,40.336,-35.299
C00603=1013.291,-74.751,-111.487,-27.653,40.255,-35.322
C00604=1013.294,-74.511,-111.507,-27.643,40.175,-35.345
C00605=1013.296,-74.271,-111.526,-27.632,40.096,-35.367
C00606=1013.299,-74.031,-111.546,-27.622,40.016,-35.390
C00607=1013.301,-73.791,-111.566,-27.612,39.936,-35.412
C00608=1013.304,-73.551,-111.585,-27.602,39.857,-35.436
C00609=1013.306,-73.311,-111.605,-27.592,39.779,-35.459
C00610=1013.308,-73.070,-111.624,-27.581,39.700,-35.481
C00611=1013.311,-72.830,-111.644,-27.571,39.623,-35.502
C00612=1013.313,-72.590,-111.663,-27.561,39.544,-35.525
C00613=1013.316,-72.349,-111.683,-27.551,39.467,-35.549
C00614=1013.318,-72.109,-111.703,-27.541,39.390,-35.571
C00615=1013.320,-71.869,-111.722,-27.531,39.313,-35.593
C00616=1013.322,-71.628,-111.742,-27.521,39.237,-35.615
C00617=1013.324,-71.387,-111.762,-27.511,39.161,-35.638
C00618=1013.327,-71.146,-111.781,-27.500,39.085,-35.660
C00619=1013.329,-70.906,-111.801,-27.490,39.009,-35.683
C00620=1013.332,-70.666,-111.820,-27.480,38.934,-35.705
C00621=1013.334,-70.425,-111.839,-27.470,38.859,-35.726
C00622=1013.336,-70.184,-111.859,-27.460,38.785,-35.749
C00623=1013.339,-69.925,-111.881,-27.450,38.705,-35.773
C00624=1013.341,-69.693,-111.900,-27.440,38.633,-35.795
C00625=1013.343,-69.462,-111.918,-27.430,38.563,-35.815
C00626=1013.346,-69.221,-111.938,-27.421,38.490,-35.837
C00627=1013.348,-68.982,-111.958,-27.411,38.416,-35.859
C00628=1013.350,-68.740,-111.977,-27.401,38.344,-35.881
C00629=1013.352,-68.500,-111.997,-27.391,38.272,-35.903
C00630=1013.355,-68.259,-112.017,-27.381,38.200,-35.925
C00631=1013.357,-68.018,-112.036,-27.371,38.128,-35.947
C00632=1013.359,-67.778,-112.055,-27.361,38.057,-35.968
C00633=1013.361,-67.537,-112.075,-27.352,37.986,-35.991
C00634=1013.364,-67.297,-112.095,-27.342,37.915,-36.012
C00635=1013.365,-67.057,-112.115,-27.332,37.845,-36.034
C00636=1013.367,-66.816,-112.134,-27.322,37.774,-36.055
C00637=1013.369,-66.576,-112.153,-27.313,37.704,-36.077
C00638=1013.372,-66.335,-112.173,-27.303,37.636,-36.098
C00639=1013.374,-66.095,-112.193,-27.293,37.566,-36.119
C00640=1013.375,-65.855,-112.212,-27.284,37.498,-36.140
C00641=1013.379,-65.615,-112.231,-27.274,37.429,-36.162
C00642=1013.380,-65.375,-112.251,-27.265,37.361,-36.183
C00643=1013.383,-65.136,-112.271,-27.255,37.294,-36.204
C00644=1013.384,-64.896,-112.291,-27.246,37.227,-36.225
C00645=1013.387,-64.656,-112.310,-27.236,37.159,-36.246
C00646=1013.388,-64.417,-112.329,-27.227,37.093,-36.267
C00647=1013.390,-64.178,-112.349,-27.217,37.027,-36.288
C00648=1013.393,-63.938,-112.368,-27.208,36.961,-36.309
C00649=1013.394,-63.700,-112.388,-27.198,36.895,-36.330
C00650=1013.397,-63.461,-112.408,-27.189,36.831,-36.350
C00651=1013.399,-63.222,-112.427,-27.180,36.765,-36.371
C00652=1013.401,-62.983,-112.446,-27.170,36.701,-36.391
C00653=1013.403,-62.745,-112.465,-27.161,36.637,-36.412
C00654=1013.405,-62.507,-112.485,-27.152,36.573,-36.432
C00655=1013.407,-62.268,-112.504,-27.143,36.509,-36.453
C00656=1013.409,-62.031,-112.523,-27.133,36.446,-36.473
C00657=1013.411,-61.793,-112.543,-27.124,36.383,-36.492
C00658=1013.413,-61.556,-112.562,-27.115,36.322,-36.512
C00659=1013.415,-61.318,-112.581,-27.106,36.259,-36.532
C00660=1013.417,-61.081,-112.601,-27.097,36.197,-36.552
C00661=1013.419,-60.844,-112.620,-27.088,36.136,-36.572
C00662=1013.420,-60.607,-112.639,-27.079,36.075,-36.591
C00663=1013.422,-60.370,-112.659,-27.070,36.014,-36.611
C00664=1013.424,-60.134,-112.677,-27.061,35.954,-36.632
C00665=1013.426,-59.897,-112.697,-27.052,35.895,-36.650
C00666=1013.428,-59.661,-112.716,-27.043,35.835,-36.670
C00667=1013.430,-59.426,-112.736,-27.035,35.775,-36.690
C00668=1013.432,-59.190,-112.754,-27.026,35.716,-36.708
C00669=1013.434,-58.954,-112.774,-27.017,35.658,-36.727
C00670=1013.436,-58.719,-112.793,-27.008,35.600,-36.746
C00671=1013.438,-58.484,-112.812,-27.000,35.542,-36.765
C00672=1013.439,-58.249,-112.832,-26.991,35.484,-36.785
C00673=1013.442,-58.014,-112.851,-26.982,35.427,-36.803
C00674=1013.443,-57.779,-112.870,-26.974,35.370,-36.822
C00675=1013.445,-57.545,-112.889,-26.965,35.313,-36.841
C00676=1013.446,-57.311,-112.908,-26.957,35.257,-36.859
C00677=1013.448,-57.076,-112.927,-26.948,35.201,-36.878
C00678=1013.450,-56.842,-112.946,-26.940,35.146,-36.896
C00679=1013.452,-56.608,-112.965,-26.931,35.091,-36.915
C00680=1013.453,-56.374,-112.984,-26.923,35.036,-36.932
C00681=1013.455,-56.140,-113.003,-26.914,34.981,-36.950
C00682=1013.457,-55.906,-113.022,-26.906,34.927,-36.968
C00683=1013.459,-55.673,-113.040,-26.898,34.873,-36.986
C00684=1013.461,-55.439,-113.060,-26.890,34.819,-37.005
C00685=1013.462,-55.205,-113.079,-26.881,34.766,-37.023
C00686=1013.464,-54.972,-113.098,-26.873,34.712,-37.040
C00687=1013.465,-54.739,-113.118,-26.865,34.660,-37.058
C00688=1013.467,-54.504,-113.137,-26.857,34.608,-37.075
C00689=1013.469,-54.271,-113.155,-26.849,34.556,-37.093
C00690=1013.471,-54.038,-113.174,-26.841,34.503,-37.110
C00691=1013.472,-53.804,-113.193,-26.832,34.451,-37.128
C00692=1013.474,-53.570,-113.212,-26.824,34.401,-37.145
C00693=1013.476,-53.337,-113.232,-26.816,34.348,-37.162
C00694=1013.477,-53.103,-113.250,-26.808,34.298,-37.179
C00695=1013.478,-52.870,-113.270,-26.800,34.248,-37.196
C00696=1013.480,-52.635,-113.289,-26.793,34.197,-37.213
C00697=1013.483,-52.402,-113.307,-26.785,34.147,-37.230
C00698=1013.484,-52.168,-113.326,-26.777,34.097,-37.248
C00699=1013.485,-51.935,-113.345,-26.769,34.048,-37.264
C00700=1013.487,-51.701,-113.364,-26.761,33.998,-37.281
C00701=1013.489,-51.468,-113.384,-26.753,33.950,-37.297
C00702=1013.490,-51.234,-113.402,-26.746,33.901,-37.314
C00703=1013.491,-51.001,-113.422,-26.738,33.853,-37.331
C00704=1013.493,-50.767,-113.440,-26.730,33.805,-37.347
C00705=1013.495,-50.533,-113.460,-26.723,33.758,-37.363
C00706=1013.496,-50.299,-113.479,-26.715,33.710,-37.379
C00707=1013.498,-50.066,-113.498,-26.707,33.663,-37.395
C00708=1013.499,-49.832,-113.517,-26.700,33.616,-37.411
C00709=1013.501,-49.598,-113.537,-26.692,33.570,-37.427
C00710=1013.502,-49.364,-113.555,-26.685,33.524,-37.443
C00711=1013.504,-49.130,-113.574,-26.677,33.477,-37.459
C00712=1013.505,-48.897,-113.593,-26.670,33.433,-37.474
C00713=1013.506,-48.663,-113.612,-26.663,33.386,-37.490
C00714=1013.508,-48.430,-113.632,-26.655,33.341,-37.505
C00715=1013.509,-48.195,-113.651,-26.648,33.297,-37.520
C00716=1013.510,-47.962,-113.670,-26.641,33.252,-37.535
C00717=1013.512,-47.728,-113.689,-26.634,33.208,-37.551
C00718=1013.514,-47.494,-113.708,-26.626,33.163,-37.566
C00719=1013.515,-47.261,-113.727,-26.619,33.120,-37.581
C00720=1013.516,-47.027,-113.746,-26.612,33.077,-37.595
C00721=1013.518,-46.688,-113.773,-26.602,33.014,-37.618
C00722=1013.520,-46.325,-113.803,-26.591,32.948,-37.641
C00723=1013.522,-46.092,-113.823,-26.584,32.906,-37.656
C00724=1013.523,-45.858,-113.841,-26.577,32.864,-37.669
C00725=1013.524,-45.624,-113.860,-26.570,32.822,-37.684
C00726=1013.526,-45.390,-113.880,-26.563,32.781,-37.698
C00727=1013.527,-45.156,-113.899,-26.557,32.739,-37.712
C00728=1013.528,-44.922,-113.918,-26.550,32.699,-37.726
C00729=1013.530,-44.689,-113.937,-26.543,32.658,-37.740
C00730=1013.532,-44.455,-113.956,-26.536,32.617,-37.754
C00731=1013.532,-44.220,-113.975,-26.530,32.577,-37.769
C00732=1013.534,-43.987,-113.995,-26.523,32.538,-37.782
C00733=1013.535,-43.753,-114.014,-26.516,32.498,-37.796
C00734=1013.537,-43.519,-114.032,-26.510,32.458,-37.809
C00735=1013.537,-43.285,-114.052,-26.503,32.419,-37.823
C00736=1013.539,-43.052,-114.071,-26.497,32.380,-37.836
C00737=1013.541,-42.817,-114.090,-26.490,32.341,-37.850
C00738=1013.541,-42.583,-114.109,-26.484,32.304,-37.862
C00739=1013.542,-42.349,-114.128,-26.477,32.265,-37.876
C00740=1013.544,-42.115,-114.148,-26.471,32.228,-37.889
C00741=1013.545,-41.881,-114.167,-26.465,32.191,-37.901
C00742=1013.546,-41.647,-114.185,-26.459,32.154,-37.914
C00743=1013.547,-41.413,-114.205,-26.452,32.117,-37.927
C00744=1013.549,-41.179,-114.224,-26.446,32.080,-37.940
C00745=1013.549,-40.945,-114.244,-26.440,32.044,-37.952
C00746=1013.551,-40.711,-114.262,-26.434,32.008,-37.965
C00747=1013.552,-40.477,-114.281,-26.428,31.973,-37.977
C00748=1013.553,-40.243,-114.300,-26.422,31.937,-37.989
C00749=1013.554,-40.009,-114.320,-26.416,31.901,-38.000
C00750=1013.556,-39.774,-114.339,-26.410,31.867,-38.013
C00751=1013.557,-39.541,-114.358,-26.404,31.832,-38.025
C00752=1013.557,-39.307,-114.377,-26.398,31.797,-38.038
C00753=1013.559,-39.073,-114.396,-26.392,31.763,-38.049
C00754=1013.560,-38.838,-114.416,-26.386,31.729,-38.061
C00755=1013.560,-38.604,-114.436,-26.380,31.695,-38.072
C00756=1013.562,-38.371,-114.454,-26.375,31.662,-38.084
C00757=1013.563,-38.136,-114.474,-26.369,31.629,-38.096
C00758=1013.564,-37.902,-114.492,-26.363,31.596,-38.106
C00759=1013.564,-37.668,-114.512,-26.358,31.563,-38.117
C00760=1013.566,-37.433,-114.531,-26.352,31.530,-38.129
C00761=1013.567,-37.199,-114.550,-26.347,31.499,-38.140
C00762=1013.568,-36.966,-114.570,-26.341,31.466,-38.150
C00763=1013.569,-36.731,-114.589,-26.336,31.435,-38.161
C00764=1013.570,-36.497,-114.608,-26.330,31.404,-38.172
C00765=1013.571,-36.263,-114.627,-26.325,31.373,-38.183
C00766=1013.572,-36.029,-114.646,-26.320,31.342,-38.193
C00767=1013.573,-35.794,-114.666,-26.314,31.311,-38.203
C00768=1013.574,-35.560,-114.684,-26.309,31.281,-38.213
C00769=1013.575,-35.326,-114.703,-26.304,31.251,-38.223
C00770=1013.576,-35.091,-114.723,-26.299,31.222,-38.233
C00771=1013.576,-34.858,-114.743,-26.294,31.192,-38.243
C00772=1013.578,-34.624,-114.762,-26.289,31.163,-38.254
C00773=1013.578,-34.390,-114.781,-26.283,31.133,-38.264
C00774=1013.579,-34.155,-114.800,-26.278,31.105,-38.273
C00775=1013.581,-33.921,-114.819,-26.273,31.076,-38.283
C00776=1013.581,-33.687,-114.838,-26.269,31.048,-38.293
C00777=1013.582,-33.452,-114.858,-26.264,31.020,-38.302
C00778=1013.583,-33.218,-114.877,-26.259,30.992,-38.311
C00779=1013.584,-32.984,-114.896,-26.254,30.965,-38.321
C00780=1013.584,-32.750,-114.915,-26.249,30.938,-38.329
C00781=1013.586,-32.516,-114.935,-26.245,30.911,-38.339
C00782=1013.586,-32.282,-114.955,-26.240,30.884,-38.347
C00783=1013.587,-32.048,-114.974,-26.235,30.858,-38.355
C00784=1013.588,-31.814,-114.993,-26.230,30.831,-38.365
C00785=1013.589,-31.579,-115.012,-26.226,30.805,-38.374
C00786=1013.590,-31.345,-115.031,-26.222,30.780,-38.381
C00787=1013.590,-31.111,-115.051,-26.217,30.754,-38.390
C00788=1013.591,-30.877,-115.070,-26.213,30.729,-38.399
C00789=1013.591,-30.642,-115.089,-26.208,30.704,-38.406
C00790=1013.593,-30.408,-115.108,-26.204,30.679,-38.414
C00791=1013.594,-30.174,-115.128,-26.200,30.655,-38.422
C00792=1013.594,-29.940,-115.147,-26.196,30.631,-38.430
C00793=1013.595,-29.706,-115.167,-26.191,30.607,-38.438
C00794=1013.595,-29.472,-115.186,-26.187,30.583,-38.446
C00795=1013.596,-29.237,-115.205,-26.183,30.559,-38.454
C00796=1013.597,-29.003,-115.225,-26.179,30.536,-38.460
C00797=1013.597,-28.769,-115.244,-26.175,30.514,-38.468
C00798=1013.599,-28.535,-115.262,-26.171,30.490,-38.476
C00799=1013.599,-28.301,-115.282,-26.167,30.467,-38.483
C00800=1013.600,-28.067,-115.301,-26.163,30.446,-38.488
C00801=1013.600,-27.833,-115.321,-26.159,30.424,-38.496
C00802=1013.601,-27.599,-115.340,-26.155,30.402,-38.503
C00803=1013.602,-27.364,-115.360,-26.151,30.380,-38.509
C00804=1013.603,-27.130,-115.379,-26.148,30.359,-38.517
C00805=1013.603,-26.896,-115.398,-26.144,30.338,-38.523
C00806=1013.604,-26.662,-115.417,-26.140,30.317,-38.529
C00807=1013.604,-26.428,-115.437,-26.137,30.297,-38.536
C00808=1013.604,-26.194,-115.456,-26.133,30.276,-38.542
C00809=1013.605,-25.960,-115.476,-26.130,30.257,-38.547
C00810=1013.606,-25.726,-115.495,-26.126,30.237,-38.554
C00811=1013.606,-25.492,-115.514,-26.123,30.217,-38.559
C00812=1013.607,-25.258,-115.534,-26.119,30.197,-38.566
C00813=1013.607,-25.023,-115.553,-26.116,30.178,-38.571
C00814=1013.608,-24.789,-115.572,-26.113,30.160,-38.577
C00815=1013.608,-24.555,-115.591,-26.109,30.141,-38.583
C00816=1013.609,-24.322,-115.611,-26.106,30.123,-38.587
C00817=1013.610,-24.088,-115.630,-26.103,30.104,-38.593
C00818=1013.610,-23.853,-115.650,-26.100,30.087,-38.597
C00819=1013.611,-23.619,-115.669,-26.096,30.069,-38.603
C00820=1013.611,-23.385,-115.688,-26.094,30.052,-38.608
C00821=1013.612,-23.151,-115.707,-26.091,30.035,-38.613
C00822=1013.612,-22.917,-115.727,-26.088,30.018,-38.618
C00823=1013.613,-22.683,-115.747,-26.085,30.001,-38.622
C00824=1013.613,-22.449,-115.766,-26.082,29.985,-38.626
C00825=1013.613,-22.215,-115.786,-26.079,29.968,-38.631
C00826=1013.614,-21.981,-115.805,-26.076,29.953,-38.635
C00827=1013.614,-21.747,-115.824,-26.073,29.937,-38.640
C00828=1013.615,-21.512,-115.843,-26.071,29.921,-38.644
C00829=1013.615,-21.279,-115.863,-26.068,29.906,-38.648
C00830=1013.616,-21.045,-115.883,-26.065,29.890,-38.652
C00831=1013.616,-20.811,-115.902,-26.063,29.876,-38.655
C00832=1013.616,-20.576,-115.922,-26.060,29.861,-38.659
C00833=1013.617,-20.299,-115.945,-26.057,29.844,-38.664
C00834=1013.617,-19.949,-115.974,-26.054,29.824,-38.669
C00835=1013.618,-19.688,-115.995,-26.051,29.808,-38.672
C00836=1013.618,-19.389,-116.020,-26.048,29.790,-38.677
C00837=1013.619,-19.063,-116.047,-26.045,29.773,-38.681
C00838=1013.619,-18.732,-116.074,-26.042,29.755,-38.686
C00839=1013.619,-18.415,-116.101,-26.039,29.738,-38.689
C00840=1013.620,-18.130,-116.124,-26.036,29.722,-38.693
C00841=1013.620,-17.883,-116.145,-26.034,29.710,-38.695
C00842=1013.620,-17.652,-116.165,-26.032,29.699,-38.697
C00843=1013.620,-17.421,-116.184,-26.030,29.687,-38.700
C00844=1013.621,-17.187,-116.203,-26.028,29.675,-38.702
C00845=1013.621,-16.950,-116.222,-26.026,29.665,-38.704
C00846=1013.622,-16.712,-116.243,-26.024,29.654,-38.706
C00847=1013.621,-16.477,-116.262,-26.023,29.644,-38.708
C00848=1013.622,-16.242,-116.282,-26.021,29.634,-38.709
C00849=1013.622,-16.007,-116.301,-26.019,29.623,-38.712
C00850=1013.622,-15.771,-116.321,-26.017,29.613,-38.714
C00851=1013.622,-15.538,-116.340,-26.016,29.603,-38.716
C00852=1013.623,-15.308,-116.359,-26.014,29.593,-38.718
C00853=1013.622,-15.082,-116.378,-26.013,29.585,-38.718
C00854=1013.623,-14.857,-116.397,-26.011,29.577,-38.719
C00855=1013.623,-14.634,-116.416,-26.010,29.568,-38.720
C00856=1013.623,-14.411,-116.434,-26.009,29.560,-38.720
C00857=1013.623,-14.187,-116.453,-26.007,29.551,-38.721
C00858=1013.624,-13.962,-116.471,-26.006,29.544,-38.721
C00859=1013.623,-13.732,-116.491,-26.005,29.536,-38.721
C00860=1013.624,-13.500,-116.510,-26.003,29.528,-38.723
C00861=1013.623,-13.262,-116.530,-26.002,29.521,-38.724
C00862=1013.624,-13.020,-116.550,-26.001,29.513,-38.725
C00863=1013.624,-12.776,-116.570,-26.000,29.507,-38.725
C00864=1013.624,-12.530,-116.591,-25.999,29.500,-38.725
C00865=1013.624,-12.284,-116.612,-25.998,29.492,-38.726
C00866=1013.624,-12.037,-116.632,-25.997,29.485,-38.726
C00867=1013.624,-11.790,-116.652,-25.995,29.479,-38.725
C00868=1013.624,-11.542,-116.674,-25.995,29.473,-38.724
C00869=1013.625,-11.294,-116.694,-25.994,29.468,-38.724
C00870=1013.625,-11.045,-116.715,-25.993,29.461,-38.724
C00871=1013.625,-10.796,-116.736,-25.992,29.456,-38.723
C00872=1013.624,-10.546,-116.757,-25.991,29.451,-38.723
C00873=1013.625,-10.296,-116.778,-25.991,29.446,-38.721
C00874=1013.624,-10.045,-116.799,-25.990,29.441,-38.720
C00875=1013.625,-9.795,-116.820,-25.989,29.437,-38.720
C00876=1013.625,-9.543,-116.841,-25.989,29.432,-38.719
C00877=1013.624,-9.292,-116.861,-25.988,29.429,-38.717
C00878=1013.625,-9.041,-116.883,-25.988,29.424,-38.717
C00879=1013.624,-8.789,-116.904,-25.987,29.421,-38.715
C00880=1013.624,-8.538,-116.925,-25.987,29.417,-38.713
C00881=1013.624,-8.286,-116.946,-25.987,29.415,-38.711
C00882=1013.624,-8.034,-116.967,-25.986,29.412,-38.710
C00883=1013.624,-7.781,-116.989,-25.986,29.409,-38.708
C00884=1013.624,-7.526,-117.010,-25.986,29.407,-38.705
C00885=1013.624,-7.271,-117.031,-25.986,29.405,-38.704
C00886=1013.624,-7.015,-117.052,-25.985,29.403,-38.701
C00887=1013.624,-6.758,-117.074,-25.985,29.402,-38.698
C00888=1013.624,-6.501,-117.096,-25.985,29.400,-38.696
C00889=1013.623,-6.243,-117.118,-25.985,29.399,-38.693
C00890=1013.623,-5.985,-117.139,-25.985,29.398,-38.691
C00891=1013.623,-5.727,-117.161,-25.986,29.398,-38.688
C00892=1013.623,-5.470,-117.182,-25.986,29.397,-38.685
C00893=1013.623,-5.218,-117.203,-25.986,29.398,-38.682
C00894=1013.622,-4.974,-117.223,-25.986,29.398,-38.678
C00895=1013.622,-4.738,-117.244,-25.987,29.398,-38.675
C00896=1013.622,-4.510,-117.263,-25.987,29.399,-38.672
C00897=1013.621,-4.285,-117.282,-25.987,29.400,-38.669
C00898=1013.621,-4.059,-117.301,-25.988,29.401,-38.665
C00899=1013.621,-3.828,-117.320,-25.988,29.401,-38.662
C00900=1013.621,-3.591,-117.340,-25.989,29.404,-38.658
C00901=1013.621,-3.349,-117.361,-25.989,29.405,-38.655
C00902=1013.621,-3.104,-117.382,-25.990,29.407,-38.651
C00903=1013.620,-2.859,-117.401,-25.991,29.409,-38.647
C00904=1013.620,-2.615,-117.422,-25.991,29.412,-38.643
C00905=1013.619,-2.372,-117.442,-25.992,29.415,-38.639
C00906=1013.620,-2.129,-117.463,-25.993,29.418,-38.633
C00907=1013.619,-1.887,-117.483,-25.994,29.421,-38.630
C00908=1013.619,-1.646,-117.503,-25.994,29.424,-38.626
C00909=1013.618,-1.406,-117.524,-25.995,29.428,-38.621
C00910=1013.618,-1.166,-117.545,-25.996,29.432,-38.616
C00911=1013.618,-0.927,-117.564,-25.997,29.435,-38.611
C00912=1013.617,-0.688,-117.585,-25.998,29.439,-38.606
C00913=1013.617,-0.451,-117.605,-25.999,29.444,-38.601
C00914=1013.617,-0.213,-117.625,-26.000,29.449,-38.597
C00915=1013.616,0.021,-117.644,-26.001,29.452,-38.592
C00916=1013.615,0.257,-117.664,-26.003,29.458,-38.586
C00917=1013.615,0.491,-117.684,-26.004,29.463,-38.581
C00918=1013.615,0.726,-117.704,-26.005,29.469,-38.576
C00919=1013.615,0.961,-117.723,-26.006,29.474,-38.571
C00920=1013.615,1.198,-117.744,-26.008,29.479,-38.565
C00921=1013.614,1.435,-117.763,-26.009,29.486,-38.560
C00922=1013.613,1.669,-117.783,-26.010,29.492,-38.554
C00923=1013.612,1.899,-117.803,-26.012,29.498,-38.549
C00924=1013.613,2.118,-117.821,-26.013,29.505,-38.543
C00925=1013.612,2.528,-117.856,-26.016,29.516,-38.532
C00926=1013.611,2.911,-117.888,-26.018,29.528,-38.522
C00927=1013.610,3.303,-117.921,-26.021,29.541,-38.512
C00928=1013.610,3.511,-117.939,-26.023,29.548,-38.505
C00929=1013.609,3.730,-117.958,-26.024,29.556,-38.500
C00930=1013.609,3.958,-117.976,-26.026,29.563,-38.493
C00931=1013.608,4.191,-117.996,-26.028,29.571,-38.487
C00932=1013.607,4.423,-118.016,-26.029,29.580,-38.479
C00933=1013.607,4.655,-118.036,-26.031,29.589,-38.473
C00934=1013.606,4.886,-118.055,-26.033,29.598,-38.466
C00935=1013.606,5.118,-118.075,-26.035,29.607,-38.460
C00936=1013.606,5.350,-118.094,-26.037,29.616,-38.453
C00937=1013.605,5.583,-118.114,-26.039,29.626,-38.445
C00938=1013.604,5.817,-118.134,-26.041,29.636,-38.438
C00939=1013.604,6.051,-118.154,-26.043,29.645,-38.431
C00940=1013.603,6.285,-118.173,-26.045,29.656,-38.423
C00941=1013.602,6.517,-118.193,-26.047,29.666,-38.416
C00942=1013.602,6.749,-118.213,-26.049,29.677,-38.409
C00943=1013.601,6.977,-118.232,-26.052,29.687,-38.400
C00944=1013.601,7.205,-118.252,-26.054,29.697,-38.394
C00945=1013.601,7.431,-118.271,-26.056,29.709,-38.385
C00946=1013.600,7.656,-118.290,-26.058,29.720,-38.377
C00947=1013.599,7.880,-118.309,-26.061,29.731,-38.369
C00948=1013.599,8.104,-118.328,-26.063,29.742,-38.362
C00949=1013.598,8.327,-118.347,-26.065,29.754,-38.355
C00950=1013.597,8.549,-118.366,-26.067,29.765,-38.347
C00951=1013.596,8.771,-118.385,-26.070,29.776,-38.339
C00952=1013.596,8.993,-118.404,-26.072,29.789,-38.330
C00953=1013.595,9.216,-118.422,-26.075,29.801,-38.322
C00954=1013.594,9.439,-118.441,-26.077,29.814,-38.314
C00955=1013.593,9.662,-118.460,-26.080,29.826,-38.305
C00956=1013.593,9.886,-118.479,-26.082,29.839,-38.298
C00957=1013.592,10.110,-118.498,-26.085,29.851,-38.289
C00958=1013.592,10.335,-118.517,-26.087,29.865,-38.280
C00959=1013.591,10.559,-118.536,-26.090,29.878,-38.271
C00960=1013.590,10.780,-118.555,-26.093,29.892,-38.263
C00961=1013.590,10.997,-118.573,-26.095,29.905,-38.254
C00962=1013.589,11.213,-118.592,-26.098,29.919,-38.245
C00963=1013.588,11.429,-118.611,-26.101,29.931,-38.236
C00964=1013.588,11.648,-118.629,-26.103,29.945,-38.228
C00965=1013.587,11.872,-118.648,-26.106,29.960,-38.218
C00966=1013.585,12.099,-118.668,-26.109,29.974,-38.210
C00967=1013.585,12.328,-118.687,-26.112,29.990,-38.201
C00968=1013.584,12.556,-118.706,-26.115,30.004,-38.191
C00969=1013.583,12.784,-118.726,-26.118,30.020,-38.181
C00970=1013.582,13.013,-118.745,-26.121,30.036,-38.171
C00971=1013.582,13.241,-118.765,-26.124,30.051,-38.161
C00972=1013.581,13.468,-118.784,-26.127,30.068,-38.152
C00973=1013.580,13.695,-118.804,-26.130,30.084,-38.142
C00974=1013.580,13.922,-118.822,-26.133,30.100,-38.133
C00975=1013.579,14.149,-118.842,-26.137,30.116,-38.122
C00976=1013.578,14.375,-118.861,-26.140,30.133,-38.112
C00977=1013.577,14.602,-118.880,-26.143,30.149,-38.103
C00978=1013.576,14.827,-118.899,-26.146,30.166,-38.092
C00979=1013.575,15.053,-118.919,-26.149,30.183,-38.082
C00980=1013.574,15.279,-118.938,-26.153,30.202,-38.071
C00981=1013.574,15.506,-118.958,-26.156,30.219,-38.061
C00982=1013.572,15.733,-118.977,-26.159,30.236,-38.051
C00983=1013.571,15.960,-118.996,-26.163,30.255,-38.039
C00984=1013.571,16.187,-119.015,-26.166,30.272,-38.028
C00985=1013.570,16.415,-119.035,-26.170,30.290,-38.018
C00986=1013.569,16.643,-119.054,-26.173,30.309,-38.007
C00987=1013.568,16.872,-119.074,-26.177,30.329,-37.996
C00988=1013.567,17.102,-119.094,-26.181,30.347,-37.985
C00989=1013.566,17.332,-119.113,-26.184,30.367,-37.973
C00990=1013.565,17.563,-119.133,-26.188,30.386,-37.962
C00991=1013.564,17.794,-119.153,-26.192,30.407,-37.950
C00992=1013.563,18.027,-119.173,-26.195,30.426,-37.940
C00993=1013.562,18.260,-119.193,-26.199,30.447,-37.928
C00994=1013.561,18.493,-119.212,-26.203,30.467,-37.916
C00995=1013.560,18.726,-119.233,-26.207,30.488,-37.904
C00996=1013.559,18.988,-119.255,-26.211,30.512,-37.891
C00997=1013.558,19.293,-119.281,-26.216,30.539,-37.875
C00998=1013.556,19.689,-119.314,-26.223,30.575,-37.854
C00999=1013.555,19.989,-119.340,-26.228,30.604,-37.838
C01000=1013.553,20.308,-119.368,-26.234,30.633,-37.822
C01001=1013.552,20.626,-119.395,-26.240,30.664,-37.806
C01002=1013.550,20.936,-119.421,-26.245,30.695,-37.788
C01003=1013.549,21.225,-119.446,-26.250,30.723,-37.772
C01004=1013.547,21.484,-119.469,-26.255,30.748,-37.759
C01005=1013.545,21.895,-119.504,-26.262,30.789,-37.736
C01006=1013.544,22.308,-119.538,-26.270,30.832,-37.713
C01007=1013.542,22.653,-119.568,-26.276,30.866,-37.694
C01008=1013.541,22.945,-119.593,-26.282,30.897,-37.678
C01009=1013.539,23.244,-119.619,-26.288,30.929,-37.660
C01010=1013.537,23.608,-119.650,-26.295,30.967,-37.640
C01011=1013.537,23.818,-119.667,-26.299,30.990,-37.627
C01012=1013.535,24.040,-119.687,-26.303,31.014,-37.614
C01013=1013.534,24.271,-119.707,-26.307,31.039,-37.601
C01014=1013.533,24.507,-119.727,-26.312,31.065,-37.587
C01015=1013.531,24.743,-119.748,-26.317,31.091,-37.573
C01016=1013.530,24.978,-119.767,-26.321,31.117,-37.559
C01017=1013.529,25.213,-119.788,-26.326,31.144,-37.545
C01018=1013.527,25.450,-119.808,-26.331,31.171,-37.532
C01019=1013.527,25.687,-119.828,-26.336,31.197,-37.518
C01020=1013.525,25.924,-119.848,-26.340,31.225,-37.503
C01021=1013.524,26.161,-119.869,-26.345,31.253,-37.488
C01022=1013.522,26.397,-119.890,-26.350,31.279,-37.474
C01023=1013.521,26.632,-119.909,-26.355,31.307,-37.459
C01024=1013.520,26.867,-119.930,-26.360,31.335,-37.445
C01025=1013.519,27.101,-119.950,-26.365,31.363,-37.430
C01026=1013.517,27.335,-119.970,-26.370,31.391,-37.416
C01027=1013.516,27.569,-119.989,-26.375,31.419,-37.401
C01028=1013.515,27.802,-120.010,-26.380,31.448,-37.387
C01029=1013.513,28.037,-120.030,-26.384,31.476,-37.372
C01030=1013.512,28.271,-120.050,-26.389,31.504,-37.357
C01031=1013.511,28.505,-120.071,-26.395,31.534,-37.342
C01032=1013.510,28.740,-120.091,-26.399,31.563,-37.328
C01033=1013.509,28.976,-120.111,-26.405,31.593,-37.313
C01034=1013.508,29.210,-120.131,-26.410,31.623,-37.297
C01035=1013.506,29.446,-120.152,-26.415,31.652,-37.283
C01036=1013.504,29.681,-120.171,-26.420,31.683,-37.266
C01037=1013.503,29.916,-120.192,-26.425,31.713,-37.251
C01038=1013.502,30.152,-120.211,-26.431,31.743,-37.236
C01039=1013.500,30.387,-120.232,-26.436,31.774,-37.221
C01040=1013.499,30.622,-120.252,-26.441,31.805,-37.205
C01041=1013.497,30.856,-120.272,-26.446,31.836,-37.190
C01042=1013.495,31.092,-120.292,-26.452,31.868,-37.174
C01043=1013.494,31.327,-120.313,-26.457,31.899,-37.159
C01044=1013.492,31.562,-120.333,-26.462,31.931,-37.143
C01045=1013.491,31.797,-120.354,-26.468,31.962,-37.127
C01046=1013.490,32.032,-120.373,-26.473,31.994,-37.111
C01047=1013.488,32.268,-120.394,-26.479,32.027,-37.095
C01048=1013.487,32.503,-120.414,-26.484,32.059,-37.080
C01049=1013.486,32.738,-120.434,-26.489,32.092,-37.062
C01050=1013.484,32.973,-120.455,-26.495,32.125,-37.047
C01051=1013.483,33.209,-120.475,-26.500,32.158,-37.030
C01052=1013.481,33.444,-120.496,-26.506,32.191,-37.014
C01053=1013.480,33.679,-120.515,-26.512,32.225,-36.998
C01054=1013.478,33.915,-120.536,-26.517,32.258,-36.981
C01055=1013.477,34.150,-120.556,-26.523,32.292,-36.964
C01056=1013.475,34.385,-120.576,-26.528,32.327,-36.948
C01057=1013.474,34.620,-120.597,-26.534,32.361,-36.932
C01058=1013.472,34.856,-120.616,-26.540,32.395,-36.915
C01059=1013.471,35.091,-120.637,-26.545,32.430,-36.899
C01060=1013.469,35.326,-120.657,-26.551,32.465,-36.882
C01061=1013.467,35.561,-120.677,-26.557,32.500,-36.866
C01062=1013.466,35.796,-120.698,-26.563,32.535,-36.848
C01063=1013.464,36.032,-120.718,-26.568,32.570,-36.832
C01064=1013.463,36.266,-120.738,-26.574,32.606,-36.815
C01065=1013.461,36.502,-120.759,-26.580,32.642,-36.798
C01066=1013.460,36.737,-120.778,-26.586,32.678,-36.781
C01067=1013.458,36.973,-120.799,-26.591,32.714,-36.763
C01068=1013.457,37.208,-120.819,-26.597,32.751,-36.745
C01069=1013.455,37.443,-120.840,-26.603,32.788,-36.729
C01070=1013.453,37.679,-120.860,-26.609,32.824,-36.712
C01071=1013.452,37.914,-120.880,-26.615,32.861,-36.694
C01072=1013.450,38.149,-120.901,-26.621,32.899,-36.677
C01073=1013.449,38.385,-120.921,-26.627,32.936,-36.659
C01074=1013.446,38.620,-120.941,-26.633,32.974,-36.641
C01075=1013.444,38.855,-120.962,-26.639,33.012,-36.624
C01076=1013.443,39.090,-120.981,-26.645,33.050,-36.606
C01077=1013.440,39.428,-121.011,-26.654,33.104,-36.582
C01078=1013.438,39.796,-121.043,-26.663,33.165,-36.553
C01079=1013.436,40.031,-121.064,-26.669,33.203,-36.534
C01080=1013.435,40.267,-121.083,-26.675,33.242,-36.517
C01081=1013.433,40.502,-121.104,-26.681,33.282,-36.499
C01082=1013.431,40.738,-121.125,-26.688,33.321,-36.482
C01083=1013.430,40.973,-121.144,-26.694,33.360,-36.463
C01084=1013.428,41.209,-121.165,-26.700,33.400,-36.445
C01085=1013.426,41.444,-121.186,-26.706,33.441,-36.427
C01086=1013.424,41.678,-121.205,-26.712,33.480,-36.408
C01087=1013.422,41.914,-121.225,-26.719,33.521,-36.391
C01088=1013.420,42.150,-121.246,-26.725,33.562,-36.373
C01089=1013.419,42.385,-121.266,-26.731,33.603,-36.353
C01090=1013.417,42.620,-121.286,-26.737,33.643,-36.336
C01091=1013.415,42.856,-121.307,-26.744,33.685,-36.316
C01092=1013.413,43.091,-121.328,-26.750,33.725,-36.299
C01093=1013.412,43.326,-121.347,-26.756,33.768,-36.280
C01094=1013.410,43.562,-121.368,-26.762,33.809,-36.261
C01095=1013.408,43.797,-121.389,-26.769,33.851,-36.242
C01096=1013.406,44.033,-121.409,-26.775,33.894,-36.224
C01097=1013.404,44.268,-121.428,-26.782,33.936,-36.205
C01098=1013.402,44.503,-121.449,-26.788,33.978,-36.186
C01099=1013.401,44.738,-121.470,-26.794,34.021,-36.168
C01100=1013.399,44.974,-121.490,-26.801,34.064,-36.148
C01101=1013.397,45.210,-121.510,-26.807,34.107,-36.130
C01102=1013.395,45.445,-121.530,-26.814,34.150,-36.110
C01103=1013.394,45.680,-121.551,-26.820,34.194,-36.092
C01104=1013.392,45.916,-121.571,-26.827,34.238,-36.073
C01105=1013.390,46.152,-121.592,-26.833,34.282,-36.054
C01106=1013.388,46.387,-121.612,-26.840,34.325,-36.034
C01107=1013.386,46.623,-121.633,-26.846,34.370,-36.015
C01108=1013.384,46.857,-121.652,-26.853,34.414,-35.996
C01109=1013.382,47.093,-121.673,-26.859,34.459,-35.977
C01110=1013.380,47.329,-121.693,-26.866,34.505,-35.957
C01111=1013.378,47.564,-121.714,-26.872,34.550,-35.939
C01112=1013.376,47.799,-121.734,-26.879,34.595,-35.918
C01113=1013.374,48.035,-121.755,-26.885,34.640,-35.900
C01114=1013.372,48.271,-121.775,-26.892,34.687,-35.880
C01115=1013.370,48.507,-121.795,-26.899,34.732,-35.860
C01116=1013.368,48.742,-121.816,-26.905,34.779,-35.841
C01117=1013.366,48.977,-121.836,-26.912,34.825,-35.821
C01118=1013.364,49.212,-121.856,-26.919,34.871,-35.801
C01119=1013.362,49.448,-121.876,-26.925,34.917,-35.782
C01120=1013.360,49.684,-121.896,-26.932,34.965,-35.763
C01121=1013.359,49.919,-121.917,-26.939,35.012,-35.742
C01122=1013.357,50.154,-121.938,-26.945,35.059,-35.723
C01123=1013.355,50.390,-121.958,-26.952,35.107,-35.702
C01124=1013.353,50.626,-121.978,-26.959,35.154,-35.684
C01125=1013.351,50.861,-121.999,-26.966,35.203,-35.663
C01126=1013.349,51.097,-122.019,-26.972,35.250,-35.643
C01127=1013.347,51.332,-122.040,-26.979,35.299,-35.623
C01128=1013.344,51.567,-122.060,-26.986,35.347,-35.603
C01129=1013.342,51.803,-122.080,-26.992,35.395,-35.583
C01130=1013.340,52.039,-122.101,-26.999,35.445,-35.563
C01131=1013.338,52.274,-122.121,-27.006,35.493,-35.543
C01132=1013.336,52.510,-122.141,-27.013,35.542,-35.523
C01133=1013.334,52.746,-122.161,-27.020,35.592,-35.503
C01134=1013.332,52.981,-122.183,-27.026,35.641,-35.483
C01135=1013.330,53.217,-122.203,-27.033,35.691,-35.462
C01136=1013.328,53.452,-122.223,-27.040,35.742,-35.442
C01137=1013.326,53.687,-122.243,-27.047,35.791,-35.422
C01138=1013.323,53.923,-122.264,-27.054,35.842,-35.402
C01139=1013.321,54.159,-122.284,-27.061,35.892,-35.382
C01140=1013.319,54.395,-122.305,-27.067,35.942,-35.361
C01141=1013.317,54.630,-122.325,-27.074,35.995,-35.340
C01142=1013.315,54.866,-122.345,-27.081,36.046,-35.320
C01143=1013.313,55.101,-122.366,-27.088,36.096,-35.300
C01144=1013.311,55.337,-122.387,-27.095,36.147,-35.279
C01145=1013.309,55.573,-122.407,-27.102,36.200,-35.259
C01146=1013.306,55.808,-122.427,-27.109,36.252,-35.238
C01147=1013.304,56.043,-122.447,-27.116,36.304,-35.218
C01148=1013.302,56.279,-122.467,-27.122,36.356,-35.197
C01149=1013.300,56.515,-122.488,-27.129,36.409,-35.176
C01150=1013.298,56.751,-122.509,-27.136,36.461,-35.155
C01151=1013.296,56.987,-122.529,-27.143,36.514,-35.134
C01152=1013.294,57.222,-122.549,-27.150,36.567,-35.114
C01153=1013.291,57.457,-122.569,-27.157,36.620,-35.093
C01154=1013.289,57.693,-122.589,-27.164,36.673,-35.073
C01155=1013.286,57.929,-122.610,-27.171,36.727,-35.051
C01156=1013.284,58.164,-122.631,-27.178,36.781,-35.031
C01157=1013.282,58.400,-122.652,-27.185,36.835,-35.010
C01158=1013.280,58.635,-122.672,-27.192,36.889,-34.990
C01159=1013.278,58.871,-122.692,-27.199,36.944,-34.969
C01160=1013.276,59.106,-122.712,-27.206,36.999,-34.948
C01161=1013.273,59.342,-122.733,-27.213,37.054,-34.927
C01162=1013.271,59.578,-122.753,-27.220,37.108,-34.905
C01163=1013.269,59.814,-122.774,-27.227,37.163,-34.884
C01164=1013.267,60.049,-122.794,-27.234,37.219,-34.864
C01165=1013.264,60.284,-122.814,-27.241,37.274,-34.843
C01166=1013.262,60.520,-122.835,-27.248,37.329,-34.822
C01167=1013.259,60.756,-122.855,-27.255,37.386,-34.801
C01168=1013.257,60.992,-122.875,-27.262,37.441,-34.780
C01169=1013.255,61.228,-122.896,-27.269,37.498,-34.758
C01170=1013.253,61.463,-122.916,-27.276,37.554,-34.738
C01171=1013.250,61.699,-122.937,-27.283,37.611,-34.717
C01172=1013.248,61.934,-122.957,-27.290,37.668,-34.696
C01173=1013.246,62.210,-122.981,-27.298,37.735,-34.671
C01174=1013.243,62.498,-123.006,-27.306,37.805,-34.645
C01175=1013.240,62.773,-123.030,-27.315,37.871,-34.620
C01176=1013.237,63.069,-123.055,-27.323,37.944,-34.594
C01177=1013.234,63.351,-123.080,-27.332,38.014,-34.568
C01178=1013.231,63.602,-123.102,-27.339,38.075,-34.546
C01179=1013.229,63.840,-123.123,-27.346,38.135,-34.524
C01180=1013.227,64.092,-123.144,-27.354,38.198,-34.501
C01181=1013.224,64.360,-123.167,-27.362,38.264,-34.477
C01182=1013.221,64.630,-123.190,-27.370,38.332,-34.454
C01183=1013.219,64.896,-123.213,-27.378,38.398,-34.429
C01184=1013.216,65.156,-123.236,-27.386,38.464,-34.406
C01185=1013.213,65.408,-123.257,-27.393,38.529,-34.382
C01186=1013.211,65.651,-123.278,-27.401,38.590,-34.360
C01187=1013.208,65.884,-123.299,-27.408,38.650,-34.339
C01188=1013.204,66.276,-123.333,-27.419,38.751,-34.304
C01189=1013.203,66.489,-123.351,-27.426,38.805,-34.285
C01190=1013.200,66.725,-123.372,-27.433,38.865,-34.264
C01191=1013.197,66.961,-123.392,-27.440,38.926,-34.242
C01192=1013.193,67.366,-123.427,-27.452,39.031,-34.205
C01193=1013.190,67.674,-123.454,-27.461,39.112,-34.178
C01194=1013.188,67.916,-123.474,-27.468,39.175,-34.155
C01195=1013.185,68.162,-123.495,-27.476,39.240,-34.132
C01196=1013.182,68.410,-123.517,-27.483,39.305,-34.110
C01197=1013.180,68.660,-123.539,-27.491,39.371,-34.088
C01198=1013.177,68.908,-123.560,-27.498,39.436,-34.065
C01199=1013.174,69.153,-123.581,-27.505,39.502,-34.043
C01200=1013.172,69.396,-123.602,-27.513,39.568,-34.020
C01201=1013.169,69.637,-123.624,-27.520,39.631,-33.998
C01202=1013.167,69.878,-123.644,-27.527,39.696,-33.977
C01203=1013.164,70.119,-123.665,-27.534,39.761,-33.954
C01204=1013.162,70.360,-123.686,-27.541,39.826,-33.933
C01205=1013.159,70.601,-123.707,-27.549,39.892,-33.911
C01206=1013.156,70.843,-123.727,-27.556,39.957,-33.888
C01207=1013.153,71.083,-123.748,-27.563,40.023,-33.867
C01208=1013.151,71.324,-123.769,-27.570,40.088,-33.845
C01209=1013.149,71.565,-123.790,-27.577,40.154,-33.823
C01210=1013.147,71.807,-123.811,-27.585,40.221,-33.801
C01211=1013.144,72.049,-123.832,-27.592,40.289,-33.778
C01212=1013.140,72.291,-123.852,-27.599,40.355,-33.756
C01213=1013.138,72.533,-123.873,-27.606,40.423,-33.734
C01214=1013.136,72.776,-123.894,-27.613,40.490,-33.712
C01215=1013.133,73.020,-123.916,-27.621,40.558,-33.690
C01216=1013.130,73.266,-123.937,-27.628,40.626,-33.668
C01217=1013.128,73.511,-123.958,-27.635,40.696,-33.645
C01218=1013.125,73.758,-123.979,-27.643,40.765,-33.623
C01219=1013.122,74.008,-124.001,-27.650,40.835,-33.600
C01220=1013.119,74.276,-124.024,-27.658,40.911,-33.575
C01221=1013.116,74.547,-124.048,-27.666,40.989,-33.550
C01222=1013.113,74.807,-124.069,-27.674,41.062,-33.527
C01223=1013.110,75.055,-124.091,-27.681,41.134,-33.504
C01224=1013.107,75.302,-124.112,-27.689,41.204,-33.482
C01225=1013.105,75.548,-124.133,-27.696,41.275,-33.459
C01226=1013.102,75.792,-124.155,-27.703,41.345,-33.437
C01227=1013.099,76.033,-124.175,-27.710,41.415,-33.416
C01228=1013.097,76.271,-124.196,-27.717,41.484,-33.394
C01229=1013.094,76.506,-124.216,-27.724,41.553,-33.373
C01230=1013.092,76.739,-124.236,-27.731,41.621,-33.351
C01231=1013.088,76.969,-124.256,-27.738,41.688,-33.330
C01232=1013.086,77.198,-124.276,-27.745,41.755,-33.309
C01233=1013.084,77.425,-124.296,-27.751,41.822,-33.289
C01234=1013.081,77.653,-124.315,-27.758,41.889,-33.268
C01235=1013.078,77.880,-124.335,-27.765,41.956,-33.247
C01236=1013.076,78.108,-124.354,-27.771,42.024,-33.227
C01237=1013.073,78.339,-124.375,-27.778,42.092,-33.207
C01238=1013.071,78.571,-124.394,-27.785,42.160,-33.186
C01239=1013.068,78.806,-124.415,-27.792,42.231,-33.164
C01240=1013.065,79.042,-124.435,-27.799,42.302,-33.142
C01241=1013.062,79.283,-124.455,-27.806,42.374,-33.121
C01242=1013.060,79.524,-124.477,-27.813,42.447,-33.099
C01243=1013.057,79.768,-124.498,-27.820,42.520,-33.077
C01244=1013.054,80.015,-124.518,-27.828,42.595,-33.055
C01245=1013.051,80.257,-124.539,-27.835,42.668,-33.033
C01246=1013.049,80.487,-124.559,-27.841,42.738,-33.012
C01247=1013.046,80.704,-124.578,-27.848,42.804,-32.993
C01248=1013.044,80.921,-124.596,-27.854,42.871,-32.973
C01249=1013.041,81.150,-124.616,-27.861,42.941,-32.952
C01250=1013.039,81.392,-124.637,-27.868,43.015,-32.931
C01251=1013.036,81.640,-124.658,-27.875,43.092,-32.909
C01252=1013.032,81.886,-124.680,-27.882,43.167,-32.887
C01253=1013.030,82.133,-124.701,-27.889,43.244,-32.864
C01254=1013.026,82.379,-124.722,-27.897,43.320,-32.842
C01255=1013.024,82.625,-124.743,-27.904,43.397,-32.819
C01256=1013.021,82.870,-124.764,-27.911,43.473,-32.798
C01257=1013.018,83.115,-124.786,-27.918,43.550,-32.776
C01258=1013.015,83.361,-124.807,-27.925,43.627,-32.755
C01259=1013.013,83.605,-124.828,-27.932,43.704,-32.733
C01260=1013.009,83.848,-124.849,-27.939,43.781,-32.712
C01261=1013.006,84.092,-124.869,-27.946,43.858,-32.690
C01262=1013.003,84.335,-124.891,-27.953,43.934,-32.669
C01263=1013.001,84.578,-124.912,-27.960,44.012,-32.647
C01264=1012.998,84.820,-124.932,-27.967,44.088,-32.626
C01265=1012.995,85.061,-124.952,-27.974,44.166,-32.604
C01266=1012.992,85.302,-124.973,-27.981,44.243,-32.582
C01267=1012.989,85.542,-124.994,-27.988,44.320,-32.562
C01268=1012.987,85.783,-125.014,-27.995,44.397,-32.540
C01269=1012.984,86.023,-125.036,-28.002,44.474,-32.519
C01270=1012.981,86.262,-125.056,-28.009,44.552,-32.498
C01271=1012.978,86.501,-125.076,-28.016,44.629,-32.476
C01272=1012.975,86.740,-125.097,-28.023,44.707,-32.456
C01273=1012.973,86.977,-125.118,-28.029,44.784,-32.435
C01274=1012.968,87.366,-125.151,-28.040,44.912,-32.401
C01275=1012.964,87.677,-125.178,-28.049,45.013,-32.374
C01276=1012.961,87.905,-125.197,-28.056,45.088,-32.354
C01277=1012.958,88.129,-125.216,-28.062,45.162,-32.334
C01278=1012.956,88.353,-125.236,-28.069,45.235,-32.315
C01279=1012.953,88.577,-125.255,-28.075,45.309,-32.295
C01280=1012.950,88.802,-125.274,-28.081,45.384,-32.276
C01281=1012.947,89.028,-125.294,-28.088,45.459,-32.257
C01282=1012.945,89.258,-125.313,-28.094,45.536,-32.237
C01283=1012.942,89.490,-125.333,-28.101,45.614,-32.216
C01284=1012.939,89.727,-125.353,-28.108,45.693,-32.196
C01285=1012.935,90.011,-125.378,-28.116,45.788,-32.171
C01286=1012.931,90.344,-125.406,-28.125,45.900,-32.144
C01287=1012.927,90.663,-125.433,-28.134,46.007,-32.117
C01288=1012.924,90.922,-125.457,-28.142,46.095,-32.094
C01289=1012.921,91.158,-125.476,-28.148,46.176,-32.074
C01290=1012.919,91.393,-125.496,-28.155,46.255,-32.054
C01291=1012.915,91.628,-125.516,-28.162,46.335,-32.034
C01292=1012.913,91.863,-125.536,-28.168,46.416,-32.013
C01293=1012.910,92.098,-125.556,-28.175,46.496,-31.995
C01294=1012.907,92.334,-125.577,-28.181,46.577,-31.974
C01295=1012.905,92.569,-125.597,-28.188,46.657,-31.954
C01296=1012.901,92.805,-125.618,-28.195,46.739,-31.935
C01297=1012.899,93.040,-125.637,-28.201,46.820,-31.915
C01298=1012.896,93.275,-125.657,-28.208,46.901,-31.895
C01299=1012.893,93.510,-125.678,-28.214,46.983,-31.876
C01300=1012.890,93.745,-125.698,-28.221,47.064,-31.856
C01301=1012.887,93.981,-125.717,-28.228,47.146,-31.836
C01302=1012.884,94.216,-125.738,-28.234,47.229,-31.817
C01303=1012.881,94.451,-125.758,-28.241,47.310,-31.798
C01304=1012.878,94.686,-125.778,-28.247,47.394,-31.778
C01305=1012.875,94.921,-125.798,-28.254,47.476,-31.758
C01306=1012.873,95.156,-125.818,-28.261,47.558,-31.740
C01307=1012.869,95.392,-125.839,-28.267,47.641,-31.720
C01308=1012.867,95.627,-125.858,-28.274,47.725,-31.700
C01309=1012.864,95.862,-125.878,-28.280,47.808,-31.681
C01310=1012.861,96.097,-125.899,-28.287,47.892,-31.662
C01311=1012.858,96.332,-125.919,-28.293,47.975,-31.642
C01312=1012.855,96.567,-125.939,-28.300,48.059,-31.624
C01313=1012.852,96.803,-125.959,-28.306,48.143,-31.605
C01314=1012.849,97.038,-125.979,-28.313,48.227,-31.586
C01315=1012.846,97.273,-125.999,-28.319,48.311,-31.568
C01316=1012.843,97.508,-126.019,-28.326,48.396,-31.548
C01317=1012.840,97.743,-126.039,-28.332,48.480,-31.529
C01318=1012.837,97.979,-126.060,-28.339,48.565,-31.511
C01319=1012.834,98.214,-126.079,-28.345,48.649,-31.492
C01320=1012.832,98.449,-126.099,-28.352,48.735,-31.473
C01321=1012.828,98.684,-126.120,-28.359,48.820,-31.455
C01322=1012.826,98.919,-126.140,-28.365,48.906,-31.436
C01323=1012.823,99.154,-126.159,-28.371,48.991,-31.417
C01324=1012.819,99.390,-126.180,-28.378,49.076,-31.400
C01325=1012.817,99.625,-126.200,-28.384,49.162,-31.381
C01326=1012.814,99.860,-126.220,-28.391,49.248,-31.363
C01327=1012.810,100.094,-126.240,-28.397,49.334,-31.344
C01328=1012.808,100.329,-126.260,-28.404,49.420,-31.326
C01329=1012.805,100.564,-126.280,-28.410,49.507,-31.308
C01330=1012.802,100.800,-126.300,-28.417,49.594,-31.289
C01331=1012.799,101.035,-126.320,-28.423,49.681,-31.271
C01332=1012.796,101.270,-126.339,-28.430,49.767,-31.254
C01333=1012.793,101.506,-126.360,-28.436,49.853,-31.236
C01334=1012.790,101.741,-126.380,-28.443,49.942,-31.218
C01335=1012.787,101.976,-126.400,-28.449,50.028,-31.200
C01336=1012.784,102.211,-126.420,-28.456,50.116,-31.182
C01337=1012.782,102.446,-126.440,-28.462,50.203,-31.166
C01338=1012.778,102.680,-126.460,-28.469,50.292,-31.147
C01339=1012.775,102.916,-126.480,-28.475,50.380,-31.130
C01340=1012.772,103.151,-126.499,-28.482,50.467,-31.113
C01341=1012.769,103.386,-126.519,-28.488,50.555,-31.095
C01342=1012.767,103.621,-126.539,-28.494,50.644,-31.078
C01343=1012.763,103.856,-126.560,-28.501,50.732,-31.060
C01344=1012.761,104.075,-126.578,-28.507,50.815,-31.045
C01345=1012.758,104.326,-126.600,-28.514,50.910,-31.026
C01346=1012.755,104.562,-126.620,-28.520,50.999,-31.010
C01347=1012.752,104.796,-126.640,-28.527,51.088,-30.993
C01348=1012.749,105.032,-126.659,-28.533,51.177,-30.975
C01349=1012.745,105.267,-126.680,-28.540,51.266,-30.958
C01350=1012.743,105.502,-126.700,-28.546,51.356,-30.942
C01351=1012.740,105.737,-126.720,-28.552,51.446,-30.924
C01352=1012.737,105.972,-126.739,-28.559,51.535,-30.909
C01353=1012.734,106.207,-126.760,-28.566,51.626,-30.892
C01354=1012.731,106.442,-126.780,-28.572,51.715,-30.875
C01355=1012.728,106.677,-126.799,-28.578,51.805,-30.858
C01356=1012.724,106.913,-126.819,-28.585,51.897,-30.842
C01357=1012.722,107.148,-126.839,-28.591,51.986,-30.827
C01358=1012.719,107.383,-126.859,-28.598,52.077,-30.810
C01359=1012.717,107.618,-126.879,-28.604,52.168,-30.794
C01360=1012.713,107.852,-126.899,-28.611,52.259,-30.778
C01361=1012.710,108.088,-126.919,-28.617,52.350,-30.762
C01362=1012.707,108.323,-126.938,-28.624,52.441,-30.746
C01363=1012.704,108.558,-126.958,-28.630,52.533,-30.730
C01364=1012.701,108.793,-126.979,-28.637,52.624,-30.715
C01365=1012.698,109.028,-126.999,-28.643,52.715,-30.699
C01366=1012.695,109.262,-127.018,-28.650,52.808,-30.683
C01367=1012.692,109.498,-127.038,-28.656,52.899,-30.668
C01368=1012.689,109.733,-127.058,-28.663,52.992,-30.653
C01369=1012.686,109.968,-127.078,-28.670,53.085,-30.637
C01370=1012.684,110.203,-127.098,-28.676,53.177,-30.623
C01371=1012.681,110.438,-127.118,-28.683,53.269,-30.607
C01372=1012.677,110.673,-127.138,-28.689,53.362,-30.593
C01373=1012.674,110.909,-127.157,-28.696,53.454,-30.577
C01374=1012.672,111.144,-127.177,-28.702,53.547,-30.562
C01375=1012.669,111.379,-127.197,-28.709,53.641,-30.547
C01376=1012.666,111.614,-127.218,-28.716,53.733,-30.533
C01377=1012.663,111.849,-127.238,-28.722,53.827,-30.519
C01378=1012.659,112.084,-127.257,-28.729,53.920,-30.504
C01379=1012.657,112.319,-127.277,-28.736,54.014,-30.490
C01380=1012.653,112.554,-127.297,-28.742,54.108,-30.476
C01381=1012.651,112.789,-127.317,-28.749,54.201,-30.461
C01382=1012.648,113.024,-127.337,-28.755,54.296,-30.446
C01383=1012.645,113.259,-127.356,-28.762,54.390,-30.432
C01384=1012.642,113.494,-127.376,-28.769,54.484,-30.419
C01385=1012.639,113.729,-127.396,-28.776,54.579,-30.404
C01386=1012.636,113.964,-127.416,-28.782,54.673,-30.390
C01387=1012.633,114.199,-127.436,-28.789,54.767,-30.377
C01388=1012.630,114.435,-127.455,-28.796,54.863,-30.363
C01389=1012.627,114.669,-127.475,-28.803,54.958,-30.349
C01390=1012.624,114.905,-127.496,-28.810,55.053,-30.337
C01391=1012.621,115.140,-127.515,-28.816,55.148,-30.323
C01392=1012.619,115.375,-127.535,-28.823,55.244,-30.309
C01393=1012.616,115.610,-127.555,-28.830,55.339,-30.297
C01394=1012.612,115.844,-127.574,-28.837,55.435,-30.284
C01395=1012.609,116.080,-127.595,-28.844,55.530,-30.271
C01396=1012.607,116.315,-127.615,-28.851,55.626,-30.258
C01397=1012.604,116.550,-127.634,-28.857,55.722,-30.245
C01398=1012.601,116.785,-127.654,-28.865,55.819,-30.233
C01399=1012.598,117.020,-127.674,-28.872,55.915,-30.221
C01400=1012.595,117.255,-127.693,-28.878,56.012,-30.207
C01401=1012.591,117.491,-127.713,-28.885,56.108,-30.195
C01402=1012.589,117.726,-127.733,-28.893,56.205,-30.184
C01403=1012.586,117.961,-127.753,-28.899,56.302,-30.170
C01404=1012.584,118.196,-127.773,-28.907,56.399,-30.159
C01405=1012.581,118.431,-127.792,-28.914,56.495,-30.148
C01406=1012.577,118.666,-127.812,-28.921,56.593,-30.135
C01407=1012.573,119.035,-127.843,-28.932,56.746,-30.117
C01408=1012.568,119.371,-127.872,-28.942,56.885,-30.101
C01409=1012.566,119.606,-127.891,-28.950,56.984,-30.089
C01410=1012.563,119.841,-127.911,-28.957,57.082,-30.078
C01411=1012.560,120.076,-127.931,-28.964,57.179,-30.068
C01412=1012.557,120.311,-127.950,-28.972,57.277,-30.057
C01413=1012.554,120.546,-127.970,-28.979,57.375,-30.046
C01414=1012.551,120.782,-127.991,-28.986,57.471,-30.035
C01415=1012.548,121.017,-128.011,-28.993,57.561,-30.025
C01416=1012.546,121.252,-128.031,-28.999,57.651,-30.015
C01417=1012.543,121.487,-128.050,-29.006,57.741,-30.006
C01418=1012.541,121.722,-128.070,-29.013,57.831,-29.997
C01419=1012.538,121.957,-128.090,-29.020,57.922,-29.988
C01420=1012.535,122.192,-128.111,-29.027,58.014,-29.978
C01421=1012.532,122.427,-128.131,-29.034,58.104,-29.969
C01422=1012.529,122.662,-128.151,-29.041,58.196,-29.959
C01423=1012.527,122.897,-128.171,-29.048,58.286,-29.951
C01424=1012.525,123.133,-128.191,-29.055,58.378,-29.941
C01425=1012.522,123.368,-128.211,-29.062,58.468,-29.933
C01426=1012.519,123.603,-128.232,-29.069,58.561,-29.924
C01427=1012.516,123.838,-128.251,-29.076,58.652,-29.915
C01428=1012.513,124.073,-128.271,-29.083,58.744,-29.906
C01429=1012.511,124.308,-128.291,-29.091,58.836,-29.900
C01430=1012.508,124.543,-128.311,-29.098,58.928,-29.891
C01431=1012.506,124.778,-128.331,-29.106,59.020,-29.883
C01432=1012.503,125.013,-128.351,-29.113,59.112,-29.875
C01433=1012.500,125.248,-128.372,-29.120,59.205,-29.867
C01434=1012.497,125.483,-128.392,-29.128,59.298,-29.859
C01435=1012.494,125.718,-128.412,-29.135,59.390,-29.851
C01436=1012.492,125.953,-128.431,-29.143,59.483,-29.844
C01437=1012.490,126.189,-128.452,-29.150,59.576,-29.836
C01438=1012.487,126.424,-128.472,-29.158,59.669,-29.828
C01439=1012.484,126.659,-128.492,-29.165,59.762,-29.822
C01440=1012.482,126.894,-128.512,-29.173,59.856,-29.814
C01441=1012.478,127.129,-128.532,-29.181,59.949,-29.808
C01442=1012.476,127.364,-128.552,-29.189,60.043,-29.801
C01443=1012.473,127.599,-128.572,-29.196,60.137,-29.794
C01444=1012.471,127.834,-128.592,-29.205,60.231,-29.789
C01445=1012.468,128.069,-128.612,-29.212,60.324,-29.781
C01446=1012.465,128.304,-128.632,-29.221,60.419,-29.775
C01447=1012.463,128.540,-128.652,-29.229,60.513,-29.769
C01448=1012.461,128.775,-128.672,-29.237,60.608,-29.763
C01449=1012.458,129.010,-128.692,-29.245,60.702,-29.757
C01450=1012.455,129.245,-128.713,-29.253,60.796,-29.751
C01451=1012.452,129.480,-128.733,-29.261,60.891,-29.746
C01452=1012.449,129.715,-128.752,-29.269,60.986,-29.739
C01453=1012.447,129.950,-128.772,-29.278,61.081,-29.734
C01454=1012.445,130.186,-128.793,-29.287,61.176,-29.730
C01455=1012.442,130.422,-128.812,-29.295,61.272,-29.723
C01456=1012.439,130.657,-128.832,-29.304,61.367,-29.719
C01457=1012.437,130.892,-128.852,-29.312,61.463,-29.714
C01458=1012.434,131.127,-128.872,-29.321,61.558,-29.710
C01459=1012.431,131.362,-128.892,-29.330,61.654,-29.705
C01460=1012.429,131.597,-128.912,-29.339,61.749,-29.701
C01461=1012.427,131.832,-128.932,-29.348,61.845,-29.697
C01462=1012.423,132.068,-128.952,-29.356,61.941,-29.692
C01463=1012.421,132.303,-128.972,-29.365,62.037,-29.688
C01464=1012.418,132.538,-128.992,-29.375,62.133,-29.685
C01465=1012.415,132.773,-129.012,-29.384,62.229,-29.682
C01466=1012.413,133.008,-129.033,-29.393,62.325,-29.678
C01467=1012.411,133.243,-129.053,-29.403,62.422,-29.675
C01468=1012.408,133.479,-129.072,-29.412,62.518,-29.672
C01469=1012.405,133.714,-129.092,-29.422,62.615,-29.669
C01470=1012.403,133.951,-129.112,-29.431,62.713,-29.665
C01471=1012.400,134.186,-129.132,-29.441,62.809,-29.663
C01472=1012.398,134.420,-129.152,-29.450,62.906,-29.660
C01473=1012.395,134.659,-129.173,-29.460,63.004,-29.658
C01474=1012.392,134.955,-129.197,-29.473,63.127,-29.655
C01475=1012.389,135.240,-129.221,-29.485,63.244,-29.652
C01476=1012.387,135.474,-129.241,-29.495,63.340,-29.651
C01477=1012.384,135.698,-129.260,-29.505,63.433,-29.650
C01478=1012.380,136.117,-129.296,-29.523,63.607,-29.647
C01479=1012.375,136.503,-129.329,-29.540,63.767,-29.646
C01480=1012.371,136.886,-129.361,-29.558,63.927,-29.644
C01481=1012.367,137.303,-129.396,-29.576,64.101,-29.643
C01482=1012.363,137.686,-129.429,-29.594,64.260,-29.642
C01483=1012.358,138.108,-129.465,-29.614,64.437,-29.643
C01484=1012.356,138.359,-129.486,-29.626,64.541,-29.643
C01485=1012.353,138.633,-129.509,-29.640,64.656,-29.645
C01486=1012.350,138.928,-129.534,-29.654,64.779,-29.646
C01487=1012.346,139.235,-129.561,-29.670,64.908,-29.647
C01488=1012.344,139.548,-129.586,-29.685,65.040,-29.650
C01489=1012.340,139.856,-129.613,-29.701,65.170,-29.651
C01490=1012.337,140.152,-129.638,-29.717,65.294,-29.655
C01491=1012.334,140.427,-129.661,-29.731,65.409,-29.656
C01492=1012.331,140.800,-129.693,-29.750,65.567,-29.660
C01493=1012.328,140.971,-129.708,-29.760,65.641,-29.662
C01494=1012.326,141.228,-129.729,-29.774,65.748,-29.667
C01495=1012.324,141.438,-129.747,-29.785,65.837,-29.669
C01496=1012.321,141.684,-129.768,-29.799,65.941,-29.672
C01497=1012.319,141.923,-129.788,-29.812,66.042,-29.676
C01498=1012.317,142.161,-129.808,-29.825,66.143,-29.679
C01499=1012.313,142.401,-129.829,-29.840,66.245,-29.685
C01500=1012.312,142.640,-129.849,-29.853,66.346,-29.689
C01501=1012.309,142.880,-129.869,-29.867,66.448,-29.694
C01502=1012.307,143.120,-129.889,-29.882,66.551,-29.699
C01503=1012.304,143.360,-129.909,-29.896,66.653,-29.704
C01504=1012.301,143.601,-129.930,-29.911,66.755,-29.709
C01505=1012.299,143.842,-129.951,-29.925,66.859,-29.715
C01506=1012.297,144.082,-129.971,-29.940,66.961,-29.721
C01507=1012.294,144.324,-129.991,-29.956,67.064,-29.728
C01508=1012.292,144.565,-130.012,-29.971,67.167,-29.734
C01509=1012.289,144.806,-130.032,-29.986,67.271,-29.741
C01510=1012.287,145.048,-130.052,-30.002,67.374,-29.749
C01511=1012.285,145.290,-130.073,-30.018,67.477,-29.756
C01512=1012.283,145.531,-130.094,-30.034,67.581,-29.763
C01513=1012.280,145.773,-130.114,-30.050,67.685,-29.771
C01514=1012.278,146.016,-130.135,-30.067,67.789,-29.779
C01515=1012.275,146.258,-130.155,-30.084,67.893,-29.788
C01516=1012.273,146.501,-130.175,-30.100,67.998,-29.796
C01517=1012.270,146.743,-130.196,-30.117,68.102,-29.806
C01518=1012.268,146.987,-130.216,-30.135,68.207,-29.816
C01519=1012.266,147.234,-130.237,-30.153,68.314,-29.825
C01520=1012.264,147.489,-130.259,-30.172,68.424,-29.836
C01521=1012.260,147.877,-130.292,-30.200,68.592,-29.852
C01522=1012.256,148.298,-130.327,-30.233,68.775,-29.872
C01523=1012.253,148.584,-130.351,-30.255,68.898,-29.886
C01524=1012.250,148.875,-130.376,-30.278,69.025,-29.900
C01525=1012.247,149.171,-130.401,-30.302,69.153,-29.916
C01526=1012.244,149.471,-130.426,-30.327,69.283,-29.932
C01527=1012.241,149.771,-130.452,-30.352,69.414,-29.949
C01528=1012.238,150.071,-130.477,-30.377,69.545,-29.965
C01529=1012.236,150.368,-130.502,-30.403,69.673,-29.984
C01530=1012.234,150.660,-130.527,-30.428,69.801,-30.001
C01531=1012.231,150.946,-130.552,-30.453,69.926,-30.019
C01532=1012.228,151.225,-130.574,-30.478,70.048,-30.037
C01533=1012.226,151.496,-130.597,-30.504,70.166,-30.056
C01534=1012.223,151.759,-130.620,-30.528,70.281,-30.073
C01535=1012.221,152.014,-130.641,-30.551,70.391,-30.090
C01536=1012.218,152.263,-130.662,-30.575,70.501,-30.108
C01537=1012.216,152.507,-130.683,-30.599,70.608,-30.127
C01538=1012.214,152.749,-130.703,-30.622,70.714,-30.143
C01539=1012.212,152.990,-130.724,-30.647,70.820,-30.163
C01540=1012.210,153.232,-130.744,-30.671,70.926,-30.181
C01541=1012.208,153.474,-130.764,-30.697,71.032,-30.202
C01542=1012.206,153.715,-130.785,-30.722,71.139,-30.221
C01543=1012.203,153.957,-130.805,-30.747,71.245,-30.241
C01544=1012.202,154.197,-130.826,-30.774,71.351,-30.263
C01545=1012.199,154.438,-130.846,-30.800,71.457,-30.284
C01546=1012.197,154.679,-130.867,-30.826,71.563,-30.306
C01547=1012.195,154.919,-130.887,-30.854,71.669,-30.329
C01548=1012.193,155.159,-130.907,-30.881,71.775,-30.351
C01549=1012.191,155.399,-130.927,-30.908,71.881,-30.374
C01550=1012.189,155.639,-130.948,-30.936,71.988,-30.397
C01551=1012.187,155.878,-130.967,-30.965,72.093,-30.423
C01552=1012.185,156.117,-130.988,-30.995,72.200,-30.449
C01553=1012.183,156.356,-131.008,-31.024,72.306,-30.473
C01554=1012.181,156.596,-131.028,-31.054,72.412,-30.499
C01555=1012.179,156.836,-131.049,-31.084,72.518,-30.525
C01556=1012.177,157.075,-131.069,-31.115,72.625,-30.553
C01557=1012.174,157.314,-131.089,-31.146,72.731,-30.580
C01558=1012.172,157.552,-131.109,-31.178,72.837,-30.607
C01559=1012.171,157.790,-131.129,-31.211,72.943,-30.637
C01560=1012.169,158.027,-131.149,-31.243,73.049,-30.666
C01561=1012.167,158.264,-131.169,-31.276,73.153,-30.695
C01562=1012.165,158.499,-131.189,-31.309,73.259,-30.725
C01563=1012.164,158.735,-131.209,-31.344,73.364,-30.758
C01564=1012.162,158.971,-131.229,-31.378,73.469,-30.787
C01565=1012.159,159.207,-131.249,-31.413,73.574,-30.819
C01566=1012.157,159.443,-131.269,-31.448,73.680,-30.852
C01567=1012.155,159.677,-131.288,-31.485,73.785,-30.887
C01568=1012.154,159.910,-131.308,-31.521,73.888,-30.920
C01569=1012.152,160.141,-131.330,-31.540,73.940,-30.938
C01570=1012.151,160.376,-131.355,-31.543,73.950,-30.940
C01571=1012.151,160.616,-131.380,-31.546,73.960,-30.943
C01572=1012.150,160.866,-131.405,-31.550,73.970,-30.947
C01573=1012.149,161.129,-131.432,-31.554,73.982,-30.951
C01574=1012.148,161.406,-131.460,-31.559,73.994,-30.955
C01575=1012.147,161.699,-131.491,-31.563,74.006,-30.959
C01576=1012.146,162.002,-131.522,-31.567,74.018,-30.963
C01577=1012.145,162.308,-131.554,-31.572,74.031,-30.967
C01578=1012.144,162.600,-131.585,-31.576,74.043,-30.971
C01579=1012.143,162.907,-131.616,-31.581,74.055,-30.975
C01580=1012.143,163.201,-131.646,-31.586,74.068,-30.981
C01581=1012.142,163.465,-131.674,-31.590,74.078,-30.985
C01582=1012.141,163.702,-131.698,-31.593,74.088,-30.988
C01583=1012.140,163.922,-131.721,-31.596,74.098,-30.990
C01584=1012.139,164.257,-131.755,-31.602,74.112,-30.996
C01585=1012.137,164.532,-131.784,-31.605,74.123,-30.998
C01586=1012.137,164.849,-131.817,-31.611,74.136,-31.004
C01587=1012.136,165.153,-131.848,-31.616,74.149,-31.010
C01588=1012.135,165.388,-131.873,-31.619,74.158,-31.013
C01589=1012.134,165.624,-131.897,-31.624,74.169,-31.017
C01590=1012.133,165.859,-131.921,-31.627,74.178,-31.020
C01591=1012.133,166.094,-131.946,-31.630,74.188,-31.022
C01592=1012.131,166.330,-131.970,-31.634,74.196,-31.027
C01593=1012.132,166.566,-131.995,-31.638,74.207,-31.031
C01594=1012.130,166.802,-132.019,-31.641,74.216,-31.034
C01595=1012.130,167.037,-132.044,-31.646,74.227,-31.038
C01596=1012.129,167.273,-132.068,-31.649,74.236,-31.041
C01597=1012.128,167.508,-132.093,-31.653,74.247,-31.045
C01598=1012.127,167.744,-132.118,-31.657,74.257,-31.050
C01599=1012.127,167.979,-132.142,-31.662,74.267,-31.054
C01600=1012.126,168.215,-132.166,-31.665,74.277,-31.057
C01601=1012.125,168.450,-132.191,-31.668,74.287,-31.059
C01602=1012.125,168.686,-132.216,-31.673,74.296,-31.065
C01603=1012.124,168.921,-132.240,-31.676,74.306,-31.068
C01604=1012.123,169.157,-132.265,-31.681,74.316,-31.073
C01605=1012.122,169.393,-132.288,-31.684,74.325,-31.075
C01606=1012.122,169.629,-132.314,-31.688,74.336,-31.080
C01607=1012.121,169.864,-132.338,-31.693,74.346,-31.084
C01608=1012.120,170.100,-132.363,-31.697,74.356,-31.089
C01609=1012.119,170.335,-132.386,-31.701,74.367,-31.093
C01610=1012.119,170.571,-132.412,-31.704,74.376,-31.096
C01611=1012.118,170.807,-132.436,-31.709,74.387,-31.100
C01612=1012.117,171.042,-132.461,-31.712,74.396,-31.103
C01613=1012.116,171.279,-132.486,-31.716,74.407,-31.108
C01614=1012.116,171.514,-132.510,-31.721,74.415,-31.112
C01615=1012.115,171.749,-132.534,-31.725,74.426,-31.117
C01616=1012.115,171.985,-132.559,-31.729,74.437,-31.119
C01617=1012.114,172.221,-132.584,-31.733,74.447,-31.124
C01618=1012.113,172.456,-132.608,-31.737,74.458,-31.128
C01619=1012.112,172.692,-132.633,-31.742,74.468,-31.133
C01620=1012.112,172.927,-132.657,-31.746,74.478,-31.137
C01621=1012.111,173.163,-132.682,-31.750,74.487,-31.142
C01622=1012.110,173.399,-132.707,-31.755,74.497,-31.147
C01623=1012.110,173.634,-132.732,-31.758,74.507,-31.149
C01624=1012.109,173.870,-132.756,-31.763,74.517,-31.154
C01625=1012.109,174.106,-132.781,-31.767,74.527,-31.159
C01626=1012.107,174.342,-132.805,-31.771,74.538,-31.163
C01627=1012.107,174.578,-132.831,-31.776,74.548,-31.168
C01628=1012.106,174.813,-132.855,-31.779,74.559,-31.171
C01629=1012.105,175.048,-132.880,-31.784,74.570,-31.175
C01630=1012.105,175.285,-132.904,-31.789,74.579,-31.181
C01631=1012.104,175.520,-132.929,-31.793,74.589,-31.184
C01632=1012.103,175.757,-132.954,-31.797,74.599,-31.189
C01633=1012.103,175.992,-132.978,-31.802,74.609,-31.194
C01634=1012.102,176.227,-133.004,-31.806,74.620,-31.198
C01635=1012.101,176.463,-133.028,-31.811,74.630,-31.203
C01636=1012.101,176.699,-133.053,-31.815,74.640,-31.208
C01637=1012.100,176.935,-133.077,-31.820,74.650,-31.212
C01638=1012.100,177.170,-133.102,-31.823,74.662,-31.215
C01639=1012.099,177.406,-133.126,-31.828,74.672,-31.220
C01640=1012.098,177.642,-133.152,-31.833,74.682,-31.224
C01641=1012.098,177.877,-133.176,-31.838,74.692,-31.231
C01642=1012.097,178.113,-133.201,-31.841,74.701,-31.234
C01643=1012.096,178.349,-133.226,-31.846,74.712,-31.239
C01644=1012.096,178.585,-133.250,-31.851,74.722,-31.243
C01645=1012.095,178.821,-133.275,-31.855,74.732,-31.248
C01646=1012.095,179.057,-133.301,-31.861,74.743,-31.255
C01647=1012.094,179.292,-133.325,-31.865,74.754,-31.258
C01648=1012.093,179.528,-133.350,-31.869,74.765,-31.262
C01649=1012.092,179.764,-133.375,-31.874,74.775,-31.267
C01650=1012.092,180.000,-133.399,-31.878,74.785,-31.272
C01651=1012.091,180.235,-133.424,-31.883,74.796,-31.277
C01652=1012.091,180.472,-133.449,-31.889,74.805,-31.283
C01653=1012.090,180.707,-133.474,-31.893,74.815,-31.288
C01654=1012.089,180.943,-133.498,-31.898,74.826,-31.293
C01655=1012.089,181.179,-133.524,-31.902,74.837,-31.296
C01656=1012.088,181.414,-133.549,-31.906,74.847,-31.301
C01657=1012.088,181.651,-133.573,-31.912,74.858,-31.307
C01658=1012.087,181.886,-133.598,-31.917,74.869,-31.312
C01659=1012.086,182.122,-133.624,-31.922,74.879,-31.317
C01660=1012.086,182.382,-133.651,-31.927,74.891,-31.322
C01661=1012.085,182.606,-133.674,-31.932,74.900,-31.328
C01662=1012.085,182.829,-133.698,-31.936,74.910,-31.331
C01663=1012.084,183.065,-133.722,-31.940,74.920,-31.336
C01664=1012.084,183.301,-133.748,-31.945,74.930,-31.341
C01665=1012.083,183.537,-133.773,-31.951,74.941,-31.348
C01666=1012.082,183.773,-133.797,-31.956,74.952,-31.353
C01667=1012.082,184.008,-133.822,-31.961,74.964,-31.358
C01668=1012.081,184.244,-133.848,-31.966,74.974,-31.362
C01669=1012.080,184.480,-133.872,-31.970,74.984,-31.367
C01670=1012.080,184.716,-133.898,-31.975,74.995,-31.372
C01671=1012.080,184.952,-133.922,-31.980,75.005,-31.377
C01672=1012.078,185.188,-133.947,-31.986,75.016,-31.384
C01673=1012.078,185.424,-133.972,-31.991,75.026,-31.389
C01674=1012.078,185.659,-133.997,-31.996,75.036,-31.394
C01675=1012.078,185.895,-134.023,-32.001,75.047,-31.401
C01676=1012.076,186.131,-134.047,-32.006,75.058,-31.406
C01677=1012.076,186.367,-134.072,-32.011,75.070,-31.411
C01678=1012.076,186.603,-134.097,-32.017,75.081,-31.417
C01679=1012.075,186.839,-134.122,-32.022,75.091,-31.422
C01680=1012.074,187.075,-134.147,-32.027,75.101,-31.428
C01681=1012.074,187.311,-134.173,-32.032,75.112,-31.433
C01682=1012.074,187.546,-134.197,-32.037,75.122,-31.438
C01683=1012.073,187.783,-134.222,-32.042,75.132,-31.443
C01684=1012.072,188.018,-134.247,-32.048,75.143,-31.450
C01685=1012.072,188.254,-134.273,-32.053,75.153,-31.455
C01686=1012.071,188.490,-134.298,-32.059,75.164,-31.461
C01687=1012.071,188.726,-134.322,-32.064,75.176,-31.467
C01688=1012.070,188.962,-134.347,-32.070,75.187,-31.473
C01689=1012.070,189.198,-134.373,-32.075,75.198,-31.479
C01690=1012.069,189.434,-134.398,-32.080,75.208,-31.484
C01691=1012.070,189.669,-134.423,-32.085,75.218,-31.489
C01692=1012.069,189.906,-134.448,-32.090,75.228,-31.494
C01693=1012.068,190.141,-134.473,-32.096,75.239,-31.501
C01694=1012.067,190.377,-134.499,-32.101,75.250,-31.506
C01695=1012.067,190.613,-134.524,-32.107,75.261,-31.513
C01696=1012.067,190.849,-134.549,-32.114,75.272,-31.520
C01697=1012.066,191.085,-134.574,-32.119,75.284,-31.525
C01698=1012.066,191.321,-134.599,-32.125,75.295,-31.532
C01699=1012.065,191.556,-134.624,-32.130,75.305,-31.537
C01700=1012.064,191.792,-134.650,-32.135,75.315,-31.543
C01701=1012.064,192.028,-134.674,-32.140,75.326,-31.548
C01702=1012.064,192.264,-134.700,-32.146,75.337,-31.555
C01703=1012.063,192.501,-134.725,-32.152,75.347,-31.560
C01704=1012.063,192.737,-134.750,-32.158,75.358,-31.567
C01705=1012.062,192.973,-134.776,-32.164,75.369,-31.574
C01706=1012.062,193.208,-134.800,-32.168,75.380,-31.578
C01707=1012.061,193.444,-134.826,-32.175,75.391,-31.585
C01708=1012.061,193.679,-134.851,-32.181,75.402,-31.592
C01709=1012.060,193.915,-134.876,-32.187,75.413,-31.599
C01710=1012.060,194.152,-134.901,-32.192,75.423,-31.604
C01711=1012.060,194.388,-134.926,-32.198,75.434,-31.610
C01712=1012.059,194.624,-134.952,-32.204,75.444,-31.617
C01713=1012.059,194.860,-134.977,-32.210,75.455,-31.624
C01714=1012.058,195.096,-135.002,-32.215,75.466,-31.629
C01715=1012.058,195.332,-135.028,-32.221,75.478,-31.635
C01716=1012.058,195.568,-135.053,-32.227,75.489,-31.642
C01717=1012.058,195.803,-135.078,-32.234,75.500,-31.649
C01718=1012.057,196.039,-135.104,-32.239,75.512,-31.655
C01719=1012.057,196.275,-135.129,-32.246,75.523,-31.662
C01720=1012.056,196.511,-135.155,-32.252,75.532,-31.669
C01721=1012.056,196.747,-135.180,-32.258,75.543,-31.676
C01722=1012.055,196.984,-135.205,-32.263,75.554,-31.680
C01723=1012.055,197.219,-135.230,-32.269,75.565,-31.687
C01724=1012.055,197.455,-135.255,-32.276,75.576,-31.695
C01725=1012.054,197.691,-135.281,-32.282,75.587,-31.702
C01726=1012.054,197.927,-135.306,-32.288,75.599,-31.707
C01727=1012.053,198.163,-135.331,-32.294,75.610,-31.715
C01728=1012.053,198.410,-135.358,-32.302,75.622,-31.724
C01729=1012.053,198.802,-135.400,-32.311,75.640,-31.733
C01730=1012.052,199.192,-135.442,-32.322,75.659,-31.744
C01731=1012.052,199.434,-135.469,-32.328,75.670,-31.752
C01732=1012.051,199.662,-135.493,-32.335,75.681,-31.759
C01733=1012.051,199.895,-135.518,-32.341,75.692,-31.767
C01734=1012.050,200.137,-135.544,-32.348,75.703,-31.774
C01735=1012.050,200.390,-135.571,-32.354,75.714,-31.780
C01736=1012.050,200.646,-135.598,-32.361,75.727,-31.787
C01737=1012.050,200.884,-135.624,-32.367,75.738,-31.795
C01738=1012.050,201.108,-135.649,-32.373,75.748,-31.800
C01739=1012.049,201.325,-135.672,-32.380,75.758,-31.810
C01740=1012.049,201.741,-135.716,-32.390,75.778,-31.819
C01741=1012.048,201.946,-135.739,-32.396,75.787,-31.827
C01742=1012.048,202.166,-135.762,-32.403,75.798,-31.834
C01743=1012.053,203.413,-135.899,-33.135,75.671,-33.089
C01744=1012.054,203.660,-135.927,-33.143,75.682,-33.097
C01745=1012.056,203.904,-135.952,-33.150,75.693,-33.105
C01746=1012.058,204.148,-135.980,-33.159,75.703,-33.117
C01747=1012.060,204.392,-136.006,-33.167,75.714,-33.126
C01748=1012.061,204.636,-136.032,-33.174,75.725,-33.134
C01749=1012.064,204.881,-136.059,-33.182,75.736,-33.142
C01750=1012.066,205.125,-136.086,-33.190,75.746,-33.152
C01751=1012.067,205.369,-136.112,-33.198,75.757,-33.160
C01752=1012.069,205.613,-136.139,-33.205,75.768,-33.169
C01753=1012.071,205.857,-136.165,-33.213,75.779,-33.177
C01754=1012.073,206.100,-136.191,-33.221,75.789,-33.187
C01755=1012.075,206.343,-136.218,-33.229,75.800,-33.195
C01756=1012.077,206.586,-136.244,-33.236,75.811,-33.204
C01757=1012.079,206.829,-136.271,-33.244,75.821,-33.214
C01758=1012.081,207.072,-136.297,-33.252,75.832,-33.222
C01759=1012.083,207.315,-136.323,-33.260,75.843,-33.230
C01760=1012.085,207.558,-136.350,-33.267,75.853,-33.239
C01761=1012.087,207.801,-136.377,-33.276,75.863,-33.249
C01762=1012.089,208.043,-136.403,-33.283,75.874,-33.257
C01763=1012.091,208.286,-136.430,-33.291,75.885,-33.266
C01764=1012.092,208.528,-136.456,-33.300,75.895,-33.276
C01765=1012.094,208.771,-136.483,-33.307,75.906,-33.285
C01766=1012.097,209.013,-136.508,-33.316,75.916,-33.295
C01767=1012.099,209.256,-136.536,-33.323,75.927,-33.303
C01768=1012.100,209.498,-136.562,-33.331,75.938,-33.312
C01769=1012.102,209.740,-136.589,-33.339,75.949,-33.320
C01770=1012.104,209.983,-136.615,-33.346,75.958,-33.329
C01771=1012.106,210.225,-136.642,-33.354,75.969,-33.337
C01772=1012.109,210.468,-136.668,-33.363,75.979,-33.348
C01773=1012.111,210.710,-136.695,-33.370,75.990,-33.356
C01774=1012.113,210.953,-136.721,-33.378,76.001,-33.365
C01775=1012.115,211.196,-136.747,-33.387,76.011,-33.375
C01776=1012.117,211.438,-136.775,-33.395,76.022,-33.384
C01777=1012.119,211.682,-136.801,-33.402,76.033,-33.393
C01778=1012.121,211.924,-136.827,-33.411,76.043,-33.403
C01779=1012.123,212.167,-136.854,-33.419,76.054,-33.412
